         IF ($FLAG[313] OR $TIMER_FLAG[7]) AND $OUT[4039] THEN
            PREVSTEP = $APP_INT[5]
            $APP_INT[5] = 30
         ENDIF
      ;ENDFOLD
   ;ENDFOLD
   ;FOLD SCHRITT 30 -- ROB EZ1/SP1/KE1 SZ3 -- ;%{P}%MKUKATPVW,%CSTEP,%VST_NR,%P 1:SCHRITT, 2:30, 3: ROB EZ1/SP1/KE1 SZ3
      ;FOLD ;%{H}
         Case 30
      ;ENDFOLD
      ;FOLD F312 = AUS ;%{SE}%MKUKATPVW %CVW_SPS %VBOASG %P 2:F312 = AUS, 3: BOASG
         $FLAG[312] = FALSE
      ;ENDFOLD
      ;FOLD -- KF1/KW1 Ausblasen ein -- ;%{SE}%MKUKATPVW %CVW_COM %VCOMMENT %P 2:-- KF1/KW1 Ausblasen ein --, 3: VW_COMMENT
      ;ENDFOLD
      ;FOLD A835 = (F330 + !F330 & !F331 & !F332) & !F289 ;%{SE}%MKUKATPVW %CVW_SPS %VBOASG %P 2:A835 = (F330 + !F330 & !F331 & !F332) & !F289, 3: BOASG
         $OUT[835] = ($FLAG[330] OR NOT $FLAG[330] AND NOT $FLAG[331] AND NOT $FLAG[332]) AND NOT $FLAG[289]
      ;ENDFOLD
      ;FOLD A859 = (F330 + !F330 & !F331 & !F332) & F289 ;%{SE}%MKUKATPVW %CVW_SPS %VBOASG %P 2:A859 = (F330 + !F330 & !F331 & !F332) & F289, 3: BOASG
         $OUT[859] = ($FLAG[330] OR NOT $FLAG[330] AND NOT $FLAG[331] AND NOT $FLAG[332]) AND $FLAG[289]
      ;ENDFOLD
      ;FOLD A1019 = (F330 + !F330 & !F331 & !F332) & F803 ;%{SE}%MKUKATPVW %CVW_SPS %VBOASG %P 2:A1019 = (F330 + !F330 & !F331 & !F332) & F803, 3: BOASG
         $OUT[1019] = ($FLAG[330] OR NOT $FLAG[330] AND NOT $FLAG[331] AND NOT $FLAG[332]) AND $FLAG[803]
      ;ENDFOLD
      ;FOLD Schritt 31 = A4039  ;%{SE}%MKUKATPVW %CVW_SPS %VST_CON %P 2:Schritt 31 = A4039 , 3: ST_CON
         IF $OUT[4039] THEN
            PREVSTEP = $APP_INT[5]
            $APP_INT[5] = 31
         ENDIF
      ;ENDFOLD
   ;ENDFOLD
   ;FOLD SCHRITT 31 -- ROB EZ1/SP1/KE1 SZ3 -- ;%{P}%MKUKATPVW,%CSTEP,%VST_NR,%P 1:SCHRITT, 2:31, 3: ROB EZ1/SP1/KE1 SZ3
      ;FOLD ;%{H}
         Case 31
      ;ENDFOLD
      ;FOLD -- RSK Fehlerausgabe KF1/KW1 Initiator/Motor -- ;%{SE}%MKUKATPVW %CVW_COM %VCOMMENT %P 2:-- RSK Fehlerausgabe KF1/KW1 Initiator/Motor --, 3: VW_COMMENT
      ;ENDFOLD
      ;FOLD F322 = !F313 ;%{SE}%MKUKATPVW %CVW_SPS %VBOASG %P 2:F322 = !F313, 3: BOASG
         $FLAG[322] = NOT $FLAG[313]
      ;ENDFOLD
      ;FOLD T7 ( EIN ) = STOP ;%{SE}%MKUKATPVW %CVW_SPS %VTSTOP %P 2:T7 ( EIN ) = STOP, 3: TSTOP
         VW(#SET_TIME,TRUE,7,1,0)
      ;ENDFOLD
      ;FOLD A834 = !F322 & !F289 ;%{SE}%MKUKATPVW %CVW_SPS %VBOASG %P 2:A834 = !F322 & !F289, 3: BOASG
         $OUT[834] = NOT $FLAG[322] AND NOT $FLAG[289]
      ;ENDFOLD
      ;FOLD A858 = !F322 & F289 ;%{SE}%MKUKATPVW %CVW_SPS %VBOASG %P 2:A858 = !F322 & F289, 3: BOASG
         $OUT[858] = NOT $FLAG[322] AND $FLAG[289]
      ;ENDFOLD
      ;FOLD A1018 = !F322 & F803 ;%{SE}%MKUKATPVW %CVW_SPS %VBOASG %P 2:A1018 = !F322 & F803, 3: BOASG
         $OUT[1018] = NOT $FLAG[322] AND $FLAG[803]
      ;ENDFOLD
      ;FOLD Schritt 32 = !F322 & A4039  ;%{SE}%MKUKATPVW %CVW_SPS %VST_CON %P 2:Schritt 32 = !F322 & A4039 , 3: ST_CON
         IF NOT $FLAG[322] AND $OUT[4039] THEN
            PREVSTEP = $APP_INT[5]
            $APP_INT[5] = 32
         ENDIF
      ;ENDFOLD
      ;FOLD Schritt 34 = F322 & A4039  ;%{SE}%MKUKATPVW %CVW_SPS %VST_CON %P 2:Schritt 34 = F322 & A4039 , 3: ST_CON
         IF $FLAG[322] AND $OUT[4039] THEN
            PREVSTEP = $APP_INT[5]
            $APP_INT[5] = 34
         ENDIF
      ;ENDFOLD
   ;ENDFOLD
   ;FOLD SCHRITT 32 -- ROB EZ1/SP1/KE1 SZ3 -- ;%{P}%MKUKATPVW,%CSTEP,%VST_NR,%P 1:SCHRITT, 2:32, 3: ROB EZ1/SP1/KE1 SZ3
      ;FOLD ;%{H}
         Case 32
      ;ENDFOLD
      ;FOLD F312 = AUS ;%{SE}%MKUKATPVW %CVW_SPS %VBOASG %P 2:F312 = AUS, 3: BOASG
         $FLAG[312] = FALSE
      ;ENDFOLD
      ;FOLD F313 = AUS ;%{SE}%MKUKATPVW %CVW_SPS %VBOASG %P 2:F313 = AUS, 3: BOASG
         $FLAG[313] = FALSE
      ;ENDFOLD
      ;FOLD -- Umdreh. KF setzen -- ;%{SE}%MKUKATPVW %CVW_COM %VCOMMENT %P 2:-- Umdreh. KF setzen --, 3: VW_COMMENT
      ;ENDFOLD
      ;FOLD F270 = F111 & F732 ;%{SE}%MKUKATPVW %CVW_SPS %VBOASG %P 2:F270 = F111 & F732, 3: BOASG
         $FLAG[270] = $FLAG[111] AND $FLAG[732]
      ;ENDFOLD
      ;FOLD i45 ( EIN ) = i13 ;%{SE}%MKUKATPVW %CVW_SPS %VARIASG %P 2:i45 ( EIN ) = i13, 3: ARIASG
         VW(#COUNTER,TRUE,45,$COUNT_I[13])
      ;ENDFOLD
      ;FOLD i13 ( F270 ) = i43 ;%{SE}%MKUKATPVW %CVW_SPS %VARIASG %P 2:i13 ( F270 ) = i43, 3: ARIASG
         VW(#COUNTER,$FLAG[270],13,$COUNT_I[43])
      ;ENDFOLD
      ;FOLD i1 ( EIN ) = 0 ;%{SE}%MKUKATPVW %CVW_SPS %VARIASG %P 2:i1 ( EIN ) = 0, 3: ARIASG
         VW(#COUNTER,TRUE,1,0)
      ;ENDFOLD
      ;FOLD -- Ueberwachungszeit EZ1/SP1 SZ3 schliessen -- ;%{SE}%MKUKATPVW %CVW_COM %VCOMMENT %P 2:-- Ueberwachungszeit EZ1/SP1 SZ3 schliessen --, 3: VW_COMMENT
      ;ENDFOLD
      ;FOLD T9 ( EIN ) = -40[1/10Sek] ;%{SE}%MKUKATPVW %CVW_SPS %VTASG %P 2:T9 ( EIN ) = -40[1/10Sek], 3: TASG
         VW(#SET_TIME,TRUE,9,0,-40)
      ;ENDFOLD
      ;FOLD -- Ueberwachungszeit KF1/KW1 -- ;%{SE}%MKUKATPVW %CVW_COM %VCOMMENT %P 2:-- Ueberwachungszeit KF1/KW1 --, 3: VW_COMMENT
      ;ENDFOLD
      ;FOLD T7 ( EIN ) = -40[1/10Sek] ;%{SE}%MKUKATPVW %CVW_SPS %VTASG %P 2:T7 ( EIN ) = -40[1/10Sek], 3: TASG
         VW(#SET_TIME,TRUE,7,0,-40)
      ;ENDFOLD
      ;FOLD Schritt 33 = A4039  ;%{SE}%MKUKATPVW %CVW_SPS %VST_CON %P 2:Schritt 33 = A4039 , 3: ST_CON
         IF $OUT[4039] THEN
            PREVSTEP = $APP_INT[5]
            $APP_INT[5] = 33
         ENDIF
      ;ENDFOLD
   ;ENDFOLD
   ;FOLD SCHRITT 33 -- ROB EZ1/SP1/KE1 SZ3 -- ;%{P}%MKUKATPVW,%CSTEP,%VST_NR,%P 1:SCHRITT, 2:33, 3: ROB EZ1/SP1/KE1 SZ3
      ;FOLD ;%{H}
         Case 33
      ;ENDFOLD
      ;FOLD F270 = AUS ;%{SE}%MKUKATPVW %CVW_SPS %VBOASG %P 2:F270 = AUS, 3: BOASG
         $FLAG[270] = FALSE
      ;ENDFOLD
      ;FOLD -- KF1/KW1 Ausblasen -- ;%{SE}%MKUKATPVW %CVW_COM %VCOMMENT %P 2:-- KF1/KW1 Ausblasen --, 3: VW_COMMENT
      ;ENDFOLD
      ;FOLD A835 = (F330 + F331 + !F330 & !F331 & !F332) & !F289 ;%{SE}%MKUKATPVW %CVW_SPS %VBOASG %P 2:A835 = (F330 + F331 + !F330 & !F331 & !F332) & !F289, 3: BOASG
         $OUT[835] = ($FLAG[330] OR $FLAG[331] OR NOT $FLAG[330] AND NOT $FLAG[331] AND NOT $FLAG[332]) AND NOT $FLAG[289]
      ;ENDFOLD
      ;FOLD A859 = (F330 + F331 + !F330 & !F331 & !F332) & F289 ;%{SE}%MKUKATPVW %CVW_SPS %VBOASG %P 2:A859 = (F330 + F331 + !F330 & !F331 & !F332) & F289, 3: BOASG
         $OUT[859] = ($FLAG[330] OR $FLAG[331] OR NOT $FLAG[330] AND NOT $FLAG[331] AND NOT $FLAG[332]) AND $FLAG[289]
      ;ENDFOLD
      ;FOLD A1019 = (F330 + F331 + !F330 & !F331 & !F332) & F803 ;%{SE}%MKUKATPVW %CVW_SPS %VBOASG %P 2:A1019 = (F330 + F331 + !F330 & !F331 & !F332) & F803, 3: BOASG
         $OUT[1019] = ($FLAG[330] OR $FLAG[331] OR NOT $FLAG[330] AND NOT $FLAG[331] AND NOT $FLAG[332]) AND $FLAG[803]
      ;ENDFOLD
      ;FOLD -- EZ1/SP1 SZ3 schliessen -- ;%{SE}%MKUKATPVW %CVW_COM %VCOMMENT %P 2:-- EZ1/SP1 SZ3 schliessen --, 3: VW_COMMENT
      ;ENDFOLD
      ;FOLD A717 = AUS ;%{SE}%MKUKATPVW %CVW_SPS %VBOASG %P 2:A717 = AUS, 3: BOASG
         $OUT[717] = FALSE
      ;ENDFOLD
      ;FOLD A718 = EIN ;%{SE}%MKUKATPVW %CVW_SPS %VBOASG %P 2:A718 = EIN, 3: BOASG
         $OUT[718] = TRUE
      ;ENDFOLD
      ;FOLD Schritt 34 = (!E717 & E718 + T9) & A4039  ;%{SE}%MKUKATPVW %CVW_SPS %VST_CON %P 2:Schritt 34 = (!E717 & E718 + T9) & A4039 , 3: ST_CON
         IF (NOT $IN[717] AND $IN[718] OR $TIMER_FLAG[9]) AND $OUT[4039] THEN
            PREVSTEP = $APP_INT[5]
            $APP_INT[5] = 34
         ENDIF
      ;ENDFOLD
   ;ENDFOLD
   ;FOLD SCHRITT 34 -- ROB EZ1/SP1/KE1 SZ3 -- ;%{P}%MKUKATPVW,%CSTEP,%VST_NR,%P 1:SCHRITT, 2:34, 3: ROB EZ1/SP1/KE1 SZ3
      ;FOLD ;%{H}
         Case 34
      ;ENDFOLD
      ;FOLD T9 ( EIN ) = STOP ;%{SE}%MKUKATPVW %CVW_SPS %VTSTOP %P 2:T9 ( EIN ) = STOP, 3: TSTOP
         VW(#SET_TIME,TRUE,9,1,0)
      ;ENDFOLD
      ;FOLD -- RSK Fehlerausgabe Kraftaufbau -- ;%{SE}%MKUKATPVW %CVW_COM %VCOMMENT %P 2:-- RSK Fehlerausgabe Kraftaufbau --, 3: VW_COMMENT
      ;ENDFOLD
      ;FOLD F325 = T9 ;%{SE}%MKUKATPVW %CVW_SPS %VBOASG %P 2:F325 = T9, 3: BOASG
         $FLAG[325] = $TIMER_FLAG[9]
      ;ENDFOLD
      ;FOLD -- KF1/KW1 abschalten bei Fehler -- ;%{SE}%MKUKATPVW %CVW_COM %VCOMMENT %P 2:-- KF1/KW1 abschalten bei Fehler --, 3: VW_COMMENT
      ;ENDFOLD
      ;FOLD A834 = !T7 & !T9 & !F289 ;%{SE}%MKUKATPVW %CVW_SPS %VBOASG %P 2:A834 = !T7 & !T9 & !F289, 3: BOASG
         $OUT[834] = NOT $TIMER_FLAG[7] AND NOT $TIMER_FLAG[9] AND NOT $FLAG[289]
      ;ENDFOLD
      ;FOLD A858 = !T7 & !T9 & F289 ;%{SE}%MKUKATPVW %CVW_SPS %VBOASG %P 2:A858 = !T7 & !T9 & F289, 3: BOASG
         $OUT[858] = NOT $TIMER_FLAG[7] AND NOT $TIMER_FLAG[9] AND $FLAG[289]
      ;ENDFOLD
      ;FOLD A1018 = !T7 & !T9 & F803 ;%{SE}%MKUKATPVW %CVW_SPS %VBOASG %P 2:A1018 = !T7 & !T9 & F803, 3: BOASG
         $OUT[1018] = NOT $TIMER_FLAG[7] AND NOT $TIMER_FLAG[9] AND $FLAG[803]
      ;ENDFOLD
      ;FOLD -- KF1/KW1 Ausblasen -- ;%{SE}%MKUKATPVW %CVW_COM %VCOMMENT %P 2:-- KF1/KW1 Ausblasen --, 3: VW_COMMENT
      ;ENDFOLD
      ;FOLD A835 = (F330 + F331 + !F330 & !F331 & !F332) & !T9 & !F289 ;%{SE}%MKUKATPVW %CVW_SPS %VBOASG %P 2:A835 = (F330 + F331 + !F330 & !F331 & !F332) & !T9 & !F289, 3: BOASG
         $OUT[835] = ($FLAG[330] OR $FLAG[331] OR NOT $FLAG[330] AND NOT $FLAG[331] AND NOT $FLAG[332]) AND NOT $TIMER_FLAG[9] AND NOT $FLAG[289]
      ;ENDFOLD
      ;FOLD A859 = (F330 + F331 + !F330 & !F331 & !F332) & !T9 & F289 ;%{SE}%MKUKATPVW %CVW_SPS %VBOASG %P 2:A859 = (F330 + F331 + !F330 & !F331 & !F332) & !T9 & F289, 3: BOASG
         $OUT[859] = ($FLAG[330] OR $FLAG[331] OR NOT $FLAG[330] AND NOT $FLAG[331] AND NOT $FLAG[332]) AND NOT $TIMER_FLAG[9] AND $FLAG[289]
      ;ENDFOLD
      ;FOLD A1019 = (F330 + F331 + !F330 & !F331 & !F332) & !T9 & F803 ;%{SE}%MKUKATPVW %CVW_SPS %VBOASG %P 2:A1019 = (F330 + F331 + !F330 & !F331 & !F332) & !T9 & F803, 3: BOASG
         $OUT[1019] = ($FLAG[330] OR $FLAG[331] OR NOT $FLAG[330] AND NOT $FLAG[331] AND NOT $FLAG[332]) AND NOT $TIMER_FLAG[9] AND $FLAG[803]
      ;ENDFOLD
      ;FOLD -- Warte Fraesen fertig oder Timeout -- ;%{SE}%MKUKATPVW %CVW_COM %VCOMMENT %P 2:-- Warte Fraesen fertig oder Timeout --, 3: VW_COMMENT
      ;ENDFOLD
      ;FOLD Schritt 35 = (F110 & F79 + F106 & !F287 & F78 + F108 & F287 & F78 + T7 + T9) & A4039  ;%{SE}%MKUKATPVW %CVW_SPS %VST_CON %P 2:Schritt 35 = (F110 & F79 + F106 & !F287 & F78 + F108 & F287 & F78 + T7 + T9) & A4039 , 3: ST_CON
         IF ($FLAG[110] AND $FLAG[79] OR $FLAG[106] AND NOT $FLAG[287] AND $FLAG[78] OR $FLAG[108] AND $FLAG[287] AND $FLAG[78] OR $TIMER_FLAG[7] OR $TIMER_FLAG[9]) AND $OUT[4039] THEN
            PREVSTEP = $APP_INT[5]
            $APP_INT[5] = 35
         ENDIF
      ;ENDFOLD
   ;ENDFOLD
   ;FOLD SCHRITT 35 -- ROB EZ1/SP1/KE1 SZ3 -- ;%{P}%MKUKATPVW,%CSTEP,%VST_NR,%P 1:SCHRITT, 2:35, 3: ROB EZ1/SP1/KE1 SZ3
      ;FOLD ;%{H}
         Case 35
      ;ENDFOLD
      ;FOLD -- Hilfsflag SK Programmwechsel -- ;%{SE}%MKUKATPVW %CVW_COM %VCOMMENT %P 2:-- Hilfsflag SK Programmwechsel --, 3: VW_COMMENT
      ;ENDFOLD
      ;FOLD F334 = AUS ;%{SE}%MKUKATPVW %CVW_SPS %VBOASG %P 2:F334 = AUS, 3: BOASG
         $FLAG[334] = FALSE
      ;ENDFOLD
      ;FOLD t7 ( EIN ) = STOP ;%{SE}%MKUKATPVW %CVW_SPS %VTSTOP %P 2:t7 ( EIN ) = STOP, 3: TSTOP
         VW(#SET_TIME,TRUE,7,1,0)
      ;ENDFOLD
      ;FOLD -- KF1 Ausblasen -- ;%{SE}%MKUKATPVW %CVW_COM %VCOMMENT %P 2:-- KF1 Ausblasen --, 3: VW_COMMENT
      ;ENDFOLD
      ;FOLD A835 = (F330 + F331 + F332 + !F330 & !F331 & !F332) & !F289 ;%{SE}%MKUKATPVW %CVW_SPS %VBOASG %P 2:A835 = (F330 + F331 + F332 + !F330 & !F331 & !F332) & !F289, 3: BOASG
         $OUT[835] = ($FLAG[330] OR $FLAG[331] OR $FLAG[332] OR NOT $FLAG[330] AND NOT $FLAG[331] AND NOT $FLAG[332]) AND NOT $FLAG[289]
      ;ENDFOLD
      ;FOLD A859 = (F330 + F331 + F332 + !F330 & !F331 & !F332) & F289 ;%{SE}%MKUKATPVW %CVW_SPS %VBOASG %P 2:A859 = (F330 + F331 + F332 + !F330 & !F331 & !F332) & F289, 3: BOASG
         $OUT[859] = ($FLAG[330] OR $FLAG[331] OR $FLAG[332] OR NOT $FLAG[330] AND NOT $FLAG[331] AND NOT $FLAG[332]) AND $FLAG[289]
      ;ENDFOLD
      ;FOLD A1019 = (F330 + F331 + F332 + !F330 & !F331 & !F332) & F803 ;%{SE}%MKUKATPVW %CVW_SPS %VBOASG %P 2:A1019 = (F330 + F331 + F332 + !F330 & !F331 & !F332) & F803, 3: BOASG
         $OUT[1019] = ($FLAG[330] OR $FLAG[331] OR $FLAG[332] OR NOT $FLAG[330] AND NOT $FLAG[331] AND NOT $FLAG[332]) AND $FLAG[803]
      ;ENDFOLD
      ;FOLD -- KF Ausblasen Ausschaltverzoegerung starten -- ;%{SE}%MKUKATPVW %CVW_COM %VCOMMENT %P 2:-- KF Ausblasen Ausschaltverzoegerung starten --, 3: VW_COMMENT
      ;ENDFOLD
      ;FOLD F736 = EIN ;%{SE}%MKUKATPVW %CVW_SPS %VBOASG %P 2:F736 = EIN, 3: BOASG
         $FLAG[736] = TRUE
      ;ENDFOLD
      ;FOLD -- EZ1/SP1 SZ3 oeffnen -- ;%{SE}%MKUKATPVW %CVW_COM %VCOMMENT %P 2:-- EZ1/SP1 SZ3 oeffnen --, 3: VW_COMMENT
      ;ENDFOLD
      ;FOLD A719 = AUS ;%{SE}%MKUKATPVW %CVW_SPS %VBOASG %P 2:A719 = AUS, 3: BOASG
         $OUT[719] = FALSE
      ;ENDFOLD
      ;FOLD A718 = AUS ;%{SE}%MKUKATPVW %CVW_SPS %VBOASG %P 2:A718 = AUS, 3: BOASG
         $OUT[718] = FALSE
      ;ENDFOLD
      ;FOLD A717 = EIN ;%{SE}%MKUKATPVW %CVW_SPS %VBOASG %P 2:A717 = EIN, 3: BOASG
         $OUT[717] = TRUE
      ;ENDFOLD
      ;FOLD -- RSK Sammelstoerung -- ;%{SE}%MKUKATPVW %CVW_COM %VCOMMENT %P 2:-- RSK Sammelstoerung --, 3: VW_COMMENT
      ;ENDFOLD
      ;FOLD F329 = T7 + T9 ;%{SE}%MKUKATPVW %CVW_SPS %VBOASG %P 2:F329 = T7 + T9, 3: BOASG
         $FLAG[329] = $TIMER_FLAG[7] OR $TIMER_FLAG[9]
      ;ENDFOLD
      ;FOLD -- Hilfsflag Startfraesen -- ;%{SE}%MKUKATPVW %CVW_COM %VCOMMENT %P 2:-- Hilfsflag Startfraesen --, 3: VW_COMMENT
      ;ENDFOLD
      ;FOLD F108 = (F108 & F78 + F110 & F79) & F287 ;%{SE}%MKUKATPVW %CVW_SPS %VBOASG %P 2:F108 = (F108 & F78 + F110 & F79) & F287, 3: BOASG
         $FLAG[108] = ($FLAG[108] AND $FLAG[78] OR $FLAG[110] AND $FLAG[79]) AND $FLAG[287]
      ;ENDFOLD
      ;FOLD F110 = !F130 & F110 + F130 & F287 & F110 ;%{SE}%MKUKATPVW %CVW_SPS %VBOASG %P 2:F110 = !F130 & F110 + F130 & F287 & F110, 3: BOASG
         $FLAG[110] = NOT $FLAG[130] AND $FLAG[110] OR $FLAG[130] AND $FLAG[287] AND $FLAG[110]
      ;ENDFOLD
      ;FOLD F287 = F78 + F79 & F130 ;%{SE}%MKUKATPVW %CVW_SPS %VBOASG %P 2:F287 = F78 + F79 & F130, 3: BOASG
         $FLAG[287] = $FLAG[78] OR $FLAG[79] AND $FLAG[130]
      ;ENDFOLD
      ;FOLD -- Neues Fraesprogramm und Zaehler ruecksetzen -- ;%{SE}%MKUKATPVW %CVW_COM %VCOMMENT %P 2:-- Neues Fraesprogramm und Zaehler ruecksetzen --, 3: VW_COMMENT
      ;ENDFOLD
      ;FOLD F270 = F108 & F732 ;%{SE}%MKUKATPVW %CVW_SPS %VBOASG %P 2:F270 = F108 & F732, 3: BOASG
         $FLAG[270] = $FLAG[108] AND $FLAG[732]
      ;ENDFOLD
      ;FOLD bin3 ( F732 ) = 38 ;%{SE}%MKUKATPVW %CVW_SPS %VARIASG %P 2:bin3 ( F732 ) = 38, 3: ARIASG
         VW(#BINOUT,$FLAG[732],3,38)
      ;ENDFOLD
      ;FOLD i13 ( F270 ) = i45 ;%{SE}%MKUKATPVW %CVW_SPS %VARIASG %P 2:i13 ( F270 ) = i45, 3: ARIASG
         VW(#COUNTER,$FLAG[270],13,$COUNT_I[45])
      ;ENDFOLD
      ;FOLD -- Wiederholung beim Startfraesen -- ;%{SE}%MKUKATPVW %CVW_COM %VCOMMENT %P 2:-- Wiederholung beim Startfraesen --, 3: VW_COMMENT
      ;ENDFOLD
      ;FOLD Schritt 32 = E717 & !E718 & (F78 & !F108 + F79 & F130 & !F108) & !F329 & A4039  ;%{SE}%MKUKATPVW %CVW_SPS %VST_CON %P 2:Schritt 32 = E717 & !E718 & (F78 & !F108 + F79 & F130 & !F108) & !F329 & A4039 , 3: ST_CON
         IF $IN[717] AND NOT $IN[718] AND ($FLAG[78] AND NOT $FLAG[108] OR $FLAG[79] AND $FLAG[130] AND NOT $FLAG[108]) AND NOT $FLAG[329] AND $OUT[4039] THEN
            PREVSTEP = $APP_INT[5]
            $APP_INT[5] = 32
         ENDIF
      ;ENDFOLD
      ;FOLD -- Weiter wenn Fraesen fertig -- ;%{SE}%MKUKATPVW %CVW_COM %VCOMMENT %P 2:-- Weiter wenn Fraesen fertig --, 3: VW_COMMENT
      ;ENDFOLD
      ;FOLD Schritt 36 = E717 & !E718 & (F79 & F110 & (!F130 + F108) + F78 & F108 + F329) & A4039  ;%{SE}%MKUKATPVW %CVW_SPS %VST_CON %P 2:Schritt 36 = E717 & !E718 & (F79 & F110 & (!F130 + F108) + F78 & F108 + F329) & A4039 , 3: ST_CON
         IF $IN[717] AND NOT $IN[718] AND ($FLAG[79] AND $FLAG[110] AND (NOT $FLAG[130] OR $FLAG[108]) OR $FLAG[78] AND $FLAG[108] OR $FLAG[329]) AND $OUT[4039] THEN
            PREVSTEP = $APP_INT[5]
            $APP_INT[5] = 36
         ENDIF
      ;ENDFOLD
      ;FOLD -- Weiter bei Fehler -- ;%{SE}%MKUKATPVW %CVW_COM %VCOMMENT %P 2:-- Weiter bei Fehler --, 3: VW_COMMENT
      ;ENDFOLD
      ;FOLD Schritt 38 = F325 & (E26 + E27) & A4039  ;%{SE}%MKUKATPVW %CVW_SPS %VST_CON %P 2:Schritt 38 = F325 & (E26 + E27) & A4039 , 3: ST_CON
         IF $FLAG[325] AND ($IN[26] OR $IN[27]) AND $OUT[4039] THEN
            PREVSTEP = $APP_INT[5]
            $APP_INT[5] = 38
         ENDIF
      ;ENDFOLD
   ;ENDFOLD
   ;FOLD SCHRITT 36 -- ROB EZ1/SP1/KE1 SZ3 -- ;%{P}%MKUKATPVW,%CSTEP,%VST_NR,%P 1:SCHRITT, 2:36, 3: ROB EZ1/SP1/KE1 SZ3
      ;FOLD ;%{H}
         Case 36
      ;ENDFOLD
      ;FOLD F270 = AUS ;%{SE}%MKUKATPVW %CVW_SPS %VBOASG %P 2:F270 = AUS, 3: BOASG
         $FLAG[270] = FALSE
      ;ENDFOLD
      ;FOLD A717 = AUS ;%{SE}%MKUKATPVW %CVW_SPS %VBOASG %P 2:A717 = AUS, 3: BOASG
         $OUT[717] = FALSE
      ;ENDFOLD
      ;FOLD -- KF1/KW1 abschalten -- ;%{SE}%MKUKATPVW %CVW_COM %VCOMMENT %P 2:-- KF1/KW1 abschalten --, 3: VW_COMMENT
      ;ENDFOLD
      ;FOLD A834 = AUS ;%{SE}%MKUKATPVW %CVW_SPS %VBOASG %P 2:A834 = AUS, 3: BOASG
         $OUT[834] = FALSE
      ;ENDFOLD
      ;FOLD A858 = AUS ;%{SE}%MKUKATPVW %CVW_SPS %VBOASG %P 2:A858 = AUS, 3: BOASG
         $OUT[858] = FALSE
      ;ENDFOLD
      ;FOLD A1018 = AUS ;%{SE}%MKUKATPVW %CVW_SPS %VBOASG %P 2:A1018 = AUS, 3: BOASG
         $OUT[1018] = FALSE
      ;ENDFOLD
      ;FOLD bin3 ( !F329 ) = 3 ;%{SE}%MKUKATPVW %CVW_SPS %VARIASG %P 2:bin3 ( !F329 ) = 3, 3: ARIASG
         VW(#BINOUT,NOT $FLAG[329],3,3)
      ;ENDFOLD
      ;FOLD -- Wartezeit Programmwechsel SK -- ;%{SE}%MKUKATPVW %CVW_COM %VCOMMENT %P 2:-- Wartezeit Programmwechsel SK --, 3: VW_COMMENT
      ;ENDFOLD
      ;FOLD T8 ( !F334 ) = -2[1/10Sek] ;%{SE}%MKUKATPVW %CVW_SPS %VTASG %P 2:T8 ( !F334 ) = -2[1/10Sek], 3: TASG
         VW(#SET_TIME,NOT $FLAG[334],8,0,-2)
      ;ENDFOLD
      ;FOLD -- Hilfsflag SK Programmwechsel -- ;%{SE}%MKUKATPVW %CVW_COM %VCOMMENT %P 2:-- Hilfsflag SK Programmwechsel --, 3: VW_COMMENT
      ;ENDFOLD
      ;FOLD F334 = EIN ;%{SE}%MKUKATPVW %CVW_SPS %VBOASG %P 2:F334 = EIN, 3: BOASG
         $FLAG[334] = TRUE
      ;ENDFOLD
      ;FOLD Schritt 37 = T8 & A4039  ;%{SE}%MKUKATPVW %CVW_SPS %VST_CON %P 2:Schritt 37 = T8 & A4039 , 3: ST_CON
         IF $TIMER_FLAG[8] AND $OUT[4039] THEN
            PREVSTEP = $APP_INT[5]
            $APP_INT[5] = 37
         ENDIF
      ;ENDFOLD
   ;ENDFOLD
   ;FOLD SCHRITT 37 -- ROB EZ1/SP1/KE1 SZ3 -- ;%{P}%MKUKATPVW,%CSTEP,%VST_NR,%P 1:SCHRITT, 2:37, 3: ROB EZ1/SP1/KE1 SZ3
      ;FOLD ;%{H}
         Case 37
      ;ENDFOLD
      ;FOLD -- Hilfsflag SK Programmwechsel -- ;%{SE}%MKUKATPVW %CVW_COM %VCOMMENT %P 2:-- Hilfsflag SK Programmwechsel --, 3: VW_COMMENT
      ;ENDFOLD
      ;FOLD F334 = AUS ;%{SE}%MKUKATPVW %CVW_SPS %VBOASG %P 2:F334 = AUS, 3: BOASG
         $FLAG[334] = FALSE
      ;ENDFOLD
      ;FOLD -- Quitt. Fraesen SK1 -- ;%{SE}%MKUKATPVW %CVW_COM %VCOMMENT %P 2:-- Quitt. Fraesen SK1 --, 3: VW_COMMENT
      ;ENDFOLD
      ;FOLD A786 = (!F329 & !F322 & !F830) + (F830 & A786) ;%{SE}%MKUKATPVW %CVW_SPS %VBOASG %P 2:A786 = (!F329 & !F322 & !F830) + (F830 & A786), 3: BOASG
         $OUT[786] = (NOT $FLAG[329] AND NOT $FLAG[322] AND NOT $FLAG[830]) OR ($FLAG[830] AND $OUT[786])
      ;ENDFOLD
      ;FOLD A722 = (!F329 & !F322 & F830) + (!F830 & A722) ;%{SE}%MKUKATPVW %CVW_SPS %VBOASG %P 2:A722 = (!F329 & !F322 & F830) + (!F830 & A722), 3: BOASG
         $OUT[722] = (NOT $FLAG[329] AND NOT $FLAG[322] AND $FLAG[830]) OR (NOT $FLAG[830] AND $OUT[722])
      ;ENDFOLD
      ;FOLD Schritt 38 = (!F830 & !E786 & E787 & !E788 + F830 & !E722 & E724 & !E723 + F329) & A4039  ;%{SE}%MKUKATPVW %CVW_SPS %VST_CON %P 2:Schritt 38 = (!F830 & !E786 & E787 & !E788 + F830 & !E722 & E724 & !E723 + F329) & A4039 , 3: ST_CON
         IF (NOT $FLAG[830] AND NOT $IN[786] AND $IN[787] AND NOT $IN[788] OR $FLAG[830] AND NOT $IN[722] AND $IN[724] AND NOT $IN[723] OR $FLAG[329]) AND $OUT[4039] THEN
            PREVSTEP = $APP_INT[5]
            $APP_INT[5] = 38
         ENDIF
      ;ENDFOLD
   ;ENDFOLD
   ;FOLD SCHRITT 38 -- ROB EZ1/SP1/KE1 SZ3 # Ende -- ;%{P}%MKUKATPVW,%CSTEP,%VST_NR,%P 1:SCHRITT, 2:38, 3: ROB EZ1/SP1/KE1 SZ3 # Ende
      ;FOLD ;%{H}
         Case 38
      ;ENDFOLD
      ;FOLD F270 = AUS ;%{SE}%MKUKATPVW %CVW_SPS %VBOASG %P 2:F270 = AUS, 3: BOASG
         $FLAG[270] = FALSE
      ;ENDFOLD
      ;FOLD -- KF1/KW1 Ausblasen -- ;%{SE}%MKUKATPVW %CVW_COM %VCOMMENT %P 2:-- KF1/KW1 Ausblasen --, 3: VW_COMMENT
      ;ENDFOLD
      ;FOLD A835 = (F330 + F331 + F332) & F736 ;%{SE}%MKUKATPVW %CVW_SPS %VBOASG %P 2:A835 = (F330 + F331 + F332) & F736, 3: BOASG
         $OUT[835] = ($FLAG[330] OR $FLAG[331] OR $FLAG[332]) AND $FLAG[736]
      ;ENDFOLD
      ;FOLD A859 = (F330 + F331 + F332) & F736 & F289 ;%{SE}%MKUKATPVW %CVW_SPS %VBOASG %P 2:A859 = (F330 + F331 + F332) & F736 & F289, 3: BOASG
         $OUT[859] = ($FLAG[330] OR $FLAG[331] OR $FLAG[332]) AND $FLAG[736] AND $FLAG[289]
      ;ENDFOLD
      ;FOLD A1019 = (F330 + F331 + F332) & F736 & F803 ;%{SE}%MKUKATPVW %CVW_SPS %VBOASG %P 2:A1019 = (F330 + F331 + F332) & F736 & F803, 3: BOASG
         $OUT[1019] = ($FLAG[330] OR $FLAG[331] OR $FLAG[332]) AND $FLAG[736] AND $FLAG[803]
      ;ENDFOLD
      ;FOLD F91 = (!E786 & E787 & !E788 & !F830 + !E722 & E724 & !E723 & F830) & !F322 & !F325 & !F329 ;%{SE}%MKUKATPVW %CVW_SPS %VBOASG %P 2:F91 = (!E786 & E787 & !E788 & !F830 + !E722 & E724 & !E723 & F830) & !F322 & !F325 & !F329, 3: BOASG
         $FLAG[91] = (NOT $IN[786] AND $IN[787] AND NOT $IN[788] AND NOT $FLAG[830] OR NOT $IN[722] AND $IN[724] AND NOT $IN[723] AND $FLAG[830]) AND NOT $FLAG[322] AND NOT $FLAG[325] AND NOT $FLAG[329]
      ;ENDFOLD
      ;FOLD Schritt 27 = (F322 + F325 + F329) & (E26 + E27) & A4039  ;%{SE}%MKUKATPVW %CVW_SPS %VST_CON %P 2:Schritt 27 = (F322 + F325 + F329) & (E26 + E27) & A4039 , 3: ST_CON
         IF ($FLAG[322] OR $FLAG[325] OR $FLAG[329]) AND ($IN[26] OR $IN[27]) AND $OUT[4039] THEN
            PREVSTEP = $APP_INT[5]
            $APP_INT[5] = 27
         ENDIF
      ;ENDFOLD
      ;FOLD Schritt 1 = F91 & !F322 & !F325 & !F329 & A4039  ;%{SE}%MKUKATPVW %CVW_SPS %VST_CON %P 2:Schritt 1 = F91 & !F322 & !F325 & !F329 & A4039 , 3: ST_CON
         IF $FLAG[91] AND NOT $FLAG[322] AND NOT $FLAG[325] AND NOT $FLAG[329] AND $OUT[4039] THEN
            PREVSTEP = $APP_INT[5]
            $APP_INT[5] = 1
         ENDIF
      ;ENDFOLD
   ;ENDFOLD
   ;FOLD SCHRITT 39 -- ROB EZ1/SP1/KE1 SZ4 # Start -- ;%{P}%MKUKATPVW,%CSTEP,%VST_NR,%P 1:SCHRITT, 2:39, 3: ROB EZ1/SP1/KE1 SZ4 # Start
      ;FOLD ;%{H}
         Case 39
      ;ENDFOLD
      ;FOLD -- RSK gestartet -- ;%{SE}%MKUKATPVW %CVW_COM %VCOMMENT %P 2:-- RSK gestartet --, 3: VW_COMMENT
      ;ENDFOLD
      ;FOLD F321 = AUS ;%{SE}%MKUKATPVW %CVW_SPS %VBOASG %P 2:F321 = AUS, 3: BOASG
         $FLAG[321] = FALSE
      ;ENDFOLD
      ;FOLD F322 = AUS ;%{SE}%MKUKATPVW %CVW_SPS %VBOASG %P 2:F322 = AUS, 3: BOASG
         $FLAG[322] = FALSE
      ;ENDFOLD
      ;FOLD F323 = AUS ;%{SE}%MKUKATPVW %CVW_SPS %VBOASG %P 2:F323 = AUS, 3: BOASG
         $FLAG[323] = FALSE
      ;ENDFOLD
      ;FOLD F324 = AUS ;%{SE}%MKUKATPVW %CVW_SPS %VBOASG %P 2:F324 = AUS, 3: BOASG
         $FLAG[324] = FALSE
      ;ENDFOLD
      ;FOLD F325 = AUS ;%{SE}%MKUKATPVW %CVW_SPS %VBOASG %P 2:F325 = AUS, 3: BOASG
         $FLAG[325] = FALSE
      ;ENDFOLD
      ;FOLD F327 = AUS ;%{SE}%MKUKATPVW %CVW_SPS %VBOASG %P 2:F327 = AUS, 3: BOASG
         $FLAG[327] = FALSE
      ;ENDFOLD
      ;FOLD F329 = AUS ;%{SE}%MKUKATPVW %CVW_SPS %VBOASG %P 2:F329 = AUS, 3: BOASG
         $FLAG[329] = FALSE
      ;ENDFOLD
      ;FOLD -- EZ1/SP1 SZ4 Zaehler -- ;%{SE}%MKUKATPVW %CVW_COM %VCOMMENT %P 2:-- EZ1/SP1 SZ4 Zaehler --, 3: VW_COMMENT
      ;ENDFOLD
      ;FOLD F112 = AUS ;%{SE}%MKUKATPVW %CVW_SPS %VBOASG %P 2:F112 = AUS, 3: BOASG
         $FLAG[112] = FALSE
      ;ENDFOLD
      ;FOLD F113 = AUS ;%{SE}%MKUKATPVW %CVW_SPS %VBOASG %P 2:F113 = AUS, 3: BOASG
         $FLAG[113] = FALSE
      ;ENDFOLD
      ;FOLD F114 = AUS ;%{SE}%MKUKATPVW %CVW_SPS %VBOASG %P 2:F114 = AUS, 3: BOASG
         $FLAG[114] = FALSE
      ;ENDFOLD
      ;FOLD F115 = AUS ;%{SE}%MKUKATPVW %CVW_SPS %VBOASG %P 2:F115 = AUS, 3: BOASG
         $FLAG[115] = FALSE
      ;ENDFOLD
      ;FOLD F116 = AUS ;%{SE}%MKUKATPVW %CVW_SPS %VBOASG %P 2:F116 = AUS, 3: BOASG
         $FLAG[116] = FALSE
      ;ENDFOLD
      ;FOLD F117 = AUS ;%{SE}%MKUKATPVW %CVW_SPS %VBOASG %P 2:F117 = AUS, 3: BOASG
         $FLAG[117] = FALSE
      ;ENDFOLD
      ;FOLD -- Hilfsflags Funktionstest KF Motor -- ;%{SE}%MKUKATPVW %CVW_COM %VCOMMENT %P 2:-- Hilfsflags Funktionstest KF Motor --, 3: VW_COMMENT
      ;ENDFOLD
      ;FOLD F312 = AUS ;%{SE}%MKUKATPVW %CVW_SPS %VBOASG %P 2:F312 = AUS, 3: BOASG
         $FLAG[312] = FALSE
      ;ENDFOLD
      ;FOLD F313 = AUS ;%{SE}%MKUKATPVW %CVW_SPS %VBOASG %P 2:F313 = AUS, 3: BOASG
         $FLAG[313] = FALSE
      ;ENDFOLD
      ;FOLD -- Rob. EZ1/SP1 SZ4 beim Fraesen -- ;%{SE}%MKUKATPVW %CVW_COM %VCOMMENT %P 2:-- Rob. EZ1/SP1 SZ4 beim Fraesen --, 3: VW_COMMENT
      ;ENDFOLD
      ;FOLD A116 = EIN ;%{SE}%MKUKATPVW %CVW_SPS %VBOASG %P 2:A116 = EIN, 3: BOASG
         $OUT[116] = TRUE
      ;ENDFOLD
      ;FOLD A130 = EIN ;%{SE}%MKUKATPVW %CVW_SPS %VBOASG %P 2:A130 = EIN, 3: BOASG
         $OUT[130] = TRUE
      ;ENDFOLD
      ;FOLD -- Quitt. Fraesen SK1 AUS -- ;%{SE}%MKUKATPVW %CVW_COM %VCOMMENT %P 2:-- Quitt. Fraesen SK1 AUS --, 3: VW_COMMENT
      ;ENDFOLD
      ;FOLD A786 = F830 & A786 ;%{SE}%MKUKATPVW %CVW_SPS %VBOASG %P 2:A786 = F830 & A786, 3: BOASG
         $OUT[786] = $FLAG[830] AND $OUT[786]
      ;ENDFOLD
      ;FOLD A722 = !F830 & A722 ;%{SE}%MKUKATPVW %CVW_SPS %VBOASG %P 2:A722 = !F830 & A722, 3: BOASG
         $OUT[722] = NOT $FLAG[830] AND $OUT[722]
      ;ENDFOLD
      ;FOLD -- Ueberwachungszeit KF1/KW1 -- ;%{SE}%MKUKATPVW %CVW_COM %VCOMMENT %P 2:-- Ueberwachungszeit KF1/KW1 --, 3: VW_COMMENT
      ;ENDFOLD
      ;FOLD t7 ( EIN ) = -30[1/10Sek] ;%{SE}%MKUKATPVW %CVW_SPS %VTASG %P 2:t7 ( EIN ) = -30[1/10Sek], 3: TASG
         VW(#SET_TIME,TRUE,7,0,-30)
      ;ENDFOLD
      ;FOLD Schritt 40 = A4039  ;%{SE}%MKUKATPVW %CVW_SPS %VST_CON %P 2:Schritt 40 = A4039 , 3: ST_CON
         IF $OUT[4039] THEN
            PREVSTEP = $APP_INT[5]
            $APP_INT[5] = 40
         ENDIF
      ;ENDFOLD
   ;ENDFOLD
   ;FOLD SCHRITT 40 -- ROB EZ1/SP1/KE1 SZ4 -- ;%{P}%MKUKATPVW,%CSTEP,%VST_NR,%P 1:SCHRITT, 2:40, 3: ROB EZ1/SP1/KE1 SZ4
      ;FOLD ;%{H}
         Case 40
      ;ENDFOLD
      ;FOLD -- KF1/KW1 einschalten -- ;%{SE}%MKUKATPVW %CVW_COM %VCOMMENT %P 2:-- KF1/KW1 einschalten --, 3: VW_COMMENT
      ;ENDFOLD
      ;FOLD i1 (EIN) = 0 ;%{SE}%MKUKATPVW %CVW_SPS %VARIASG %P 2:i1 (EIN) = 0, 3: ARIASG
         VW(#COUNTER,TRUE,1,0)
      ;ENDFOLD
      ;FOLD A834 = !F289 ;%{SE}%MKUKATPVW %CVW_SPS %VBOASG %P 2:A834 = !F289, 3: BOASG
         $OUT[834] = NOT $FLAG[289]
      ;ENDFOLD
      ;FOLD A858 = F289 ;%{SE}%MKUKATPVW %CVW_SPS %VBOASG %P 2:A858 = F289, 3: BOASG
         $OUT[858] = $FLAG[289]
      ;ENDFOLD
      ;FOLD A1018 = F803 ;%{SE}%MKUKATPVW %CVW_SPS %VBOASG %P 2:A1018 = F803, 3: BOASG
         $OUT[1018] = $FLAG[803]
      ;ENDFOLD
      ;FOLD Schritt 41 = A4039  ;%{SE}%MKUKATPVW %CVW_SPS %VST_CON %P 2:Schritt 41 = A4039 , 3: ST_CON
         IF $OUT[4039] THEN
            PREVSTEP = $APP_INT[5]
            $APP_INT[5] = 41
         ENDIF
      ;ENDFOLD
   ;ENDFOLD
   ;FOLD SCHRITT 41 -- ROB EZ1/SP1/KE1 SZ4 -- ;%{P}%MKUKATPVW,%CSTEP,%VST_NR,%P 1:SCHRITT, 2:41, 3: ROB EZ1/SP1/KE1 SZ4
      ;FOLD ;%{H}
         Case 41
      ;ENDFOLD
      ;FOLD -- Funktionstest KF Motor -- ;%{SE}%MKUKATPVW %CVW_COM %VCOMMENT %P 2:-- Funktionstest KF Motor --, 3: VW_COMMENT
      ;ENDFOLD
      ;FOLD F312 = EIN ;%{SE}%MKUKATPVW %CVW_SPS %VBOASG %P 2:F312 = EIN, 3: BOASG
         $FLAG[312] = TRUE
      ;ENDFOLD
      ;FOLD F313 = i1 > 2 ;%{SE}%MKUKATPVW %CVW_SPS %VBOCMP %P 2:F313 = i1 > 2, 3: BOCMP
         $FLAG[313] = $COUNT_I[1] > 2
      ;ENDFOLD
      ;FOLD Schritt 42 = (F313 + T7) & A4039  ;%{SE}%MKUKATPVW %CVW_SPS %VST_CON %P 2:Schritt 42 = (F313 + T7) & A4039 , 3: ST_CON
         IF ($FLAG[313] OR $TIMER_FLAG[7]) AND $OUT[4039] THEN
            PREVSTEP = $APP_INT[5]
            $APP_INT[5] = 42
         ENDIF
      ;ENDFOLD
   ;ENDFOLD
   ;FOLD SCHRITT 42 -- ROB EZ1/SP1/KE1 SZ4 -- ;%{P}%MKUKATPVW,%CSTEP,%VST_NR,%P 1:SCHRITT, 2:42, 3: ROB EZ1/SP1/KE1 SZ4
      ;FOLD ;%{H}
         Case 42
      ;ENDFOLD
      ;FOLD F312 = AUS ;%{SE}%MKUKATPVW %CVW_SPS %VBOASG %P 2:F312 = AUS, 3: BOASG
         $FLAG[312] = FALSE
      ;ENDFOLD
      ;FOLD -- KF1/KW1 Ausblasen ein -- ;%{SE}%MKUKATPVW %CVW_COM %VCOMMENT %P 2:-- KF1/KW1 Ausblasen ein --, 3: VW_COMMENT
      ;ENDFOLD
      ;FOLD A835 = (F330 + !F330 & !F331 & !F332) & !F289 ;%{SE}%MKUKATPVW %CVW_SPS %VBOASG %P 2:A835 = (F330 + !F330 & !F331 & !F332) & !F289, 3: BOASG
         $OUT[835] = ($FLAG[330] OR NOT $FLAG[330] AND NOT $FLAG[331] AND NOT $FLAG[332]) AND NOT $FLAG[289]
      ;ENDFOLD
      ;FOLD A859 = (F330 + !F330 & !F331 & !F332) & F289 ;%{SE}%MKUKATPVW %CVW_SPS %VBOASG %P 2:A859 = (F330 + !F330 & !F331 & !F332) & F289, 3: BOASG
         $OUT[859] = ($FLAG[330] OR NOT $FLAG[330] AND NOT $FLAG[331] AND NOT $FLAG[332]) AND $FLAG[289]
      ;ENDFOLD
      ;FOLD A1019 = (F330 + !F330 & !F331 & !F332) & F803 ;%{SE}%MKUKATPVW %CVW_SPS %VBOASG %P 2:A1019 = (F330 + !F330 & !F331 & !F332) & F803, 3: BOASG
         $OUT[1019] = ($FLAG[330] OR NOT $FLAG[330] AND NOT $FLAG[331] AND NOT $FLAG[332]) AND $FLAG[803]
      ;ENDFOLD
      ;FOLD Schritt 43 = A4039  ;%{SE}%MKUKATPVW %CVW_SPS %VST_CON %P 2:Schritt 43 = A4039 , 3: ST_CON
         IF $OUT[4039] THEN
            PREVSTEP = $APP_INT[5]
            $APP_INT[5] = 43
         ENDIF
      ;ENDFOLD
   ;ENDFOLD
   ;FOLD SCHRITT 43 -- ROB EZ1/SP1/KE1 SZ4 -- ;%{P}%MKUKATPVW,%CSTEP,%VST_NR,%P 1:SCHRITT, 2:43, 3: ROB EZ1/SP1/KE1 SZ4
      ;FOLD ;%{H}
         Case 43
      ;ENDFOLD
      ;FOLD -- RSK Fehlerausgabe KF1/KW1 Initiator/Motor -- ;%{SE}%MKUKATPVW %CVW_COM %VCOMMENT %P 2:-- RSK Fehlerausgabe KF1/KW1 Initiator/Motor --, 3: VW_COMMENT
      ;ENDFOLD
      ;FOLD F322 = !F313 ;%{SE}%MKUKATPVW %CVW_SPS %VBOASG %P 2:F322 = !F313, 3: BOASG
         $FLAG[322] = NOT $FLAG[313]
      ;ENDFOLD
      ;FOLD T7 ( EIN ) = STOP ;%{SE}%MKUKATPVW %CVW_SPS %VTSTOP %P 2:T7 ( EIN ) = STOP, 3: TSTOP
         VW(#SET_TIME,TRUE,7,1,0)
      ;ENDFOLD
      ;FOLD A834 = !F322 & !F289 ;%{SE}%MKUKATPVW %CVW_SPS %VBOASG %P 2:A834 = !F322 & !F289, 3: BOASG
         $OUT[834] = NOT $FLAG[322] AND NOT $FLAG[289]
      ;ENDFOLD
      ;FOLD A858 = !F322 & F289 ;%{SE}%MKUKATPVW %CVW_SPS %VBOASG %P 2:A858 = !F322 & F289, 3: BOASG
         $OUT[858] = NOT $FLAG[322] AND $FLAG[289]
      ;ENDFOLD
      ;FOLD A1018 = !F322 & F803 ;%{SE}%MKUKATPVW %CVW_SPS %VBOASG %P 2:A1018 = !F322 & F803, 3: BOASG
         $OUT[1018] = NOT $FLAG[322] AND $FLAG[803]
      ;ENDFOLD
      ;FOLD Schritt 44 = !F322 & A4039  ;%{SE}%MKUKATPVW %CVW_SPS %VST_CON %P 2:Schritt 44 = !F322 & A4039 , 3: ST_CON
         IF NOT $FLAG[322] AND $OUT[4039] THEN
            PREVSTEP = $APP_INT[5]
            $APP_INT[5] = 44
         ENDIF
      ;ENDFOLD
      ;FOLD Schritt 46 = F322 & A4039  ;%{SE}%MKUKATPVW %CVW_SPS %VST_CON %P 2:Schritt 46 = F322 & A4039 , 3: ST_CON
         IF $FLAG[322] AND $OUT[4039] THEN
            PREVSTEP = $APP_INT[5]
            $APP_INT[5] = 46
         ENDIF
      ;ENDFOLD
   ;ENDFOLD
   ;FOLD SCHRITT 44 -- ROB EZ1/SP1/KE1 SZ4 -- ;%{P}%MKUKATPVW,%CSTEP,%VST_NR,%P 1:SCHRITT, 2:44, 3: ROB EZ1/SP1/KE1 SZ4
      ;FOLD ;%{H}
         Case 44
      ;ENDFOLD
      ;FOLD F312 = AUS ;%{SE}%MKUKATPVW %CVW_SPS %VBOASG %P 2:F312 = AUS, 3: BOASG
         $FLAG[312] = FALSE
      ;ENDFOLD
      ;FOLD F313 = AUS ;%{SE}%MKUKATPVW %CVW_SPS %VBOASG %P 2:F313 = AUS, 3: BOASG
         $FLAG[313] = FALSE
      ;ENDFOLD
      ;FOLD -- Umdreh. KF setzen -- ;%{SE}%MKUKATPVW %CVW_COM %VCOMMENT %P 2:-- Umdreh. KF setzen --, 3: VW_COMMENT
      ;ENDFOLD
      ;FOLD F270 = F117 & F732 ;%{SE}%MKUKATPVW %CVW_SPS %VBOASG %P 2:F270 = F117 & F732, 3: BOASG
         $FLAG[270] = $FLAG[117] AND $FLAG[732]
      ;ENDFOLD
      ;FOLD i45 ( EIN ) = i16 ;%{SE}%MKUKATPVW %CVW_SPS %VARIASG %P 2:i45 ( EIN ) = i16, 3: ARIASG
         VW(#COUNTER,TRUE,45,$COUNT_I[16])
      ;ENDFOLD
      ;FOLD i16 ( F270 ) = i43 ;%{SE}%MKUKATPVW %CVW_SPS %VARIASG %P 2:i16 ( F270 ) = i43, 3: ARIASG
         VW(#COUNTER,$FLAG[270],16,$COUNT_I[43])
      ;ENDFOLD
      ;FOLD i1 ( EIN ) = 0 ;%{SE}%MKUKATPVW %CVW_SPS %VARIASG %P 2:i1 ( EIN ) = 0, 3: ARIASG
         VW(#COUNTER,TRUE,1,0)
      ;ENDFOLD
      ;FOLD -- Ueberwachungszeit EZ1/SP1/KE1 SZ4 schliessen -- ;%{SE}%MKUKATPVW %CVW_COM %VCOMMENT %P 2:-- Ueberwachungszeit EZ1/SP1/KE1 SZ4 schliessen --, 3: VW_COMMENT
      ;ENDFOLD
      ;FOLD T9 ( EIN ) = -40[1/10Sek] ;%{SE}%MKUKATPVW %CVW_SPS %VTASG %P 2:T9 ( EIN ) = -40[1/10Sek], 3: TASG
         VW(#SET_TIME,TRUE,9,0,-40)
      ;ENDFOLD
      ;FOLD -- Ueberwachungszeit KF1 -- ;%{SE}%MKUKATPVW %CVW_COM %VCOMMENT %P 2:-- Ueberwachungszeit KF1 --, 3: VW_COMMENT
      ;ENDFOLD
      ;FOLD T7 ( EIN ) = -40[1/10Sek] ;%{SE}%MKUKATPVW %CVW_SPS %VTASG %P 2:T7 ( EIN ) = -40[1/10Sek], 3: TASG
         VW(#SET_TIME,TRUE,7,0,-40)
      ;ENDFOLD
      ;FOLD Schritt 45 = A4039  ;%{SE}%MKUKATPVW %CVW_SPS %VST_CON %P 2:Schritt 45 = A4039 , 3: ST_CON
         IF $OUT[4039] THEN
            PREVSTEP = $APP_INT[5]
            $APP_INT[5] = 45
         ENDIF
      ;ENDFOLD
   ;ENDFOLD
   ;FOLD SCHRITT 45 -- ROB EZ1/SP1/KE1 SZ4 -- ;%{P}%MKUKATPVW,%CSTEP,%VST_NR,%P 1:SCHRITT, 2:45, 3: ROB EZ1/SP1/KE1 SZ4
      ;FOLD ;%{H}
         Case 45
      ;ENDFOLD
      ;FOLD F270 = AUS ;%{SE}%MKUKATPVW %CVW_SPS %VBOASG %P 2:F270 = AUS, 3: BOASG
         $FLAG[270] = FALSE
      ;ENDFOLD
      ;FOLD -- KF1/KW1 Ausblasen -- ;%{SE}%MKUKATPVW %CVW_COM %VCOMMENT %P 2:-- KF1/KW1 Ausblasen --, 3: VW_COMMENT
      ;ENDFOLD
      ;FOLD A835 = (F330 + F331 + !F330 & !F331 & !F332) & !F289 ;%{SE}%MKUKATPVW %CVW_SPS %VBOASG %P 2:A835 = (F330 + F331 + !F330 & !F331 & !F332) & !F289, 3: BOASG
         $OUT[835] = ($FLAG[330] OR $FLAG[331] OR NOT $FLAG[330] AND NOT $FLAG[331] AND NOT $FLAG[332]) AND NOT $FLAG[289]
      ;ENDFOLD
      ;FOLD A859 = (F330 + F331 + !F330 & !F331 & !F332) & F289 ;%{SE}%MKUKATPVW %CVW_SPS %VBOASG %P 2:A859 = (F330 + F331 + !F330 & !F331 & !F332) & F289, 3: BOASG
         $OUT[859] = ($FLAG[330] OR $FLAG[331] OR NOT $FLAG[330] AND NOT $FLAG[331] AND NOT $FLAG[332]) AND $FLAG[289]
      ;ENDFOLD
      ;FOLD A1019 = (F330 + F331 + !F330 & !F331 & !F332) & F803 ;%{SE}%MKUKATPVW %CVW_SPS %VBOASG %P 2:A1019 = (F330 + F331 + !F330 & !F331 & !F332) & F803, 3: BOASG
         $OUT[1019] = ($FLAG[330] OR $FLAG[331] OR NOT $FLAG[330] AND NOT $FLAG[331] AND NOT $FLAG[332]) AND $FLAG[803]
      ;ENDFOLD
      ;FOLD -- EZ1/SP1 SZ4 schliessen -- ;%{SE}%MKUKATPVW %CVW_COM %VCOMMENT %P 2:-- EZ1/SP1 SZ4 schliessen --, 3: VW_COMMENT
      ;ENDFOLD
      ;FOLD A717 = AUS ;%{SE}%MKUKATPVW %CVW_SPS %VBOASG %P 2:A717 = AUS, 3: BOASG
         $OUT[717] = FALSE
      ;ENDFOLD
      ;FOLD A718 = EIN ;%{SE}%MKUKATPVW %CVW_SPS %VBOASG %P 2:A718 = EIN, 3: BOASG
         $OUT[718] = TRUE
      ;ENDFOLD
      ;FOLD Schritt 46 = (!E717 & E718 + T9) & A4039  ;%{SE}%MKUKATPVW %CVW_SPS %VST_CON %P 2:Schritt 46 = (!E717 & E718 + T9) & A4039 , 3: ST_CON
         IF (NOT $IN[717] AND $IN[718] OR $TIMER_FLAG[9]) AND $OUT[4039] THEN
            PREVSTEP = $APP_INT[5]
            $APP_INT[5] = 46
         ENDIF
      ;ENDFOLD
   ;ENDFOLD
   ;FOLD SCHRITT 46 -- ROB EZ1/SP1/KE1 SZ4 -- ;%{P}%MKUKATPVW,%CSTEP,%VST_NR,%P 1:SCHRITT, 2:46, 3: ROB EZ1/SP1/KE1 SZ4
      ;FOLD ;%{H}
         Case 46
      ;ENDFOLD
      ;FOLD T9 ( EIN ) = STOP ;%{SE}%MKUKATPVW %CVW_SPS %VTSTOP %P 2:T9 ( EIN ) = STOP, 3: TSTOP
         VW(#SET_TIME,TRUE,9,1,0)
      ;ENDFOLD
      ;FOLD -- RSK Fehlerausgabe Kraftaufbau -- ;%{SE}%MKUKATPVW %CVW_COM %VCOMMENT %P 2:-- RSK Fehlerausgabe Kraftaufbau --, 3: VW_COMMENT
      ;ENDFOLD
      ;FOLD F325 = T9 ;%{SE}%MKUKATPVW %CVW_SPS %VBOASG %P 2:F325 = T9, 3: BOASG
         $FLAG[325] = $TIMER_FLAG[9]
      ;ENDFOLD
      ;FOLD -- KF1/KW1 abschalten bei Fehler -- ;%{SE}%MKUKATPVW %CVW_COM %VCOMMENT %P 2:-- KF1/KW1 abschalten bei Fehler --, 3: VW_COMMENT
      ;ENDFOLD
      ;FOLD A834 = !T7 & !T9 & !F289 ;%{SE}%MKUKATPVW %CVW_SPS %VBOASG %P 2:A834 = !T7 & !T9 & !F289, 3: BOASG
         $OUT[834] = NOT $TIMER_FLAG[7] AND NOT $TIMER_FLAG[9] AND NOT $FLAG[289]
      ;ENDFOLD
      ;FOLD A858 = !T7 & !T9 & F289 ;%{SE}%MKUKATPVW %CVW_SPS %VBOASG %P 2:A858 = !T7 & !T9 & F289, 3: BOASG
         $OUT[858] = NOT $TIMER_FLAG[7] AND NOT $TIMER_FLAG[9] AND $FLAG[289]
      ;ENDFOLD
      ;FOLD A1018 = !T7 & !T9 & F803 ;%{SE}%MKUKATPVW %CVW_SPS %VBOASG %P 2:A1018 = !T7 & !T9 & F803, 3: BOASG
         $OUT[1018] = NOT $TIMER_FLAG[7] AND NOT $TIMER_FLAG[9] AND $FLAG[803]
      ;ENDFOLD
      ;FOLD -- KF1/KW1 Ausblasen -- ;%{SE}%MKUKATPVW %CVW_COM %VCOMMENT %P 2:-- KF1/KW1 Ausblasen --, 3: VW_COMMENT
      ;ENDFOLD
      ;FOLD A835 = (F330 + F331 + !F330 & !F331 & !F332) & !T9 & !F289 ;%{SE}%MKUKATPVW %CVW_SPS %VBOASG %P 2:A835 = (F330 + F331 + !F330 & !F331 & !F332) & !T9 & !F289, 3: BOASG
         $OUT[835] = ($FLAG[330] OR $FLAG[331] OR NOT $FLAG[330] AND NOT $FLAG[331] AND NOT $FLAG[332]) AND NOT $TIMER_FLAG[9] AND NOT $FLAG[289]
      ;ENDFOLD
      ;FOLD A859 = (F330 + F331 + !F330 & !F331 & !F332) & !T9 & F289 ;%{SE}%MKUKATPVW %CVW_SPS %VBOASG %P 2:A859 = (F330 + F331 + !F330 & !F331 & !F332) & !T9 & F289, 3: BOASG
         $OUT[859] = ($FLAG[330] OR $FLAG[331] OR NOT $FLAG[330] AND NOT $FLAG[331] AND NOT $FLAG[332]) AND NOT $TIMER_FLAG[9] AND $FLAG[289]
      ;ENDFOLD
      ;FOLD A1019 = (F330 + F331 + !F330 & !F331 & !F332) & !T9 & F803 ;%{SE}%MKUKATPVW %CVW_SPS %VBOASG %P 2:A1019 = (F330 + F331 + !F330 & !F331 & !F332) & !T9 & F803, 3: BOASG
         $OUT[1019] = ($FLAG[330] OR $FLAG[331] OR NOT $FLAG[330] AND NOT $FLAG[331] AND NOT $FLAG[332]) AND NOT $TIMER_FLAG[9] AND $FLAG[803]
      ;ENDFOLD
      ;FOLD -- Warte Fraesen fertig oder Timeout -- ;%{SE}%MKUKATPVW %CVW_COM %VCOMMENT %P 2:-- Warte Fraesen fertig oder Timeout --, 3: VW_COMMENT
      ;ENDFOLD
      ;FOLD Schritt 47 = (F116 & F79 + F112 & !F287 & F78 + F114 & F287 & F78 + T7 + T9) & A4039  ;%{SE}%MKUKATPVW %CVW_SPS %VST_CON %P 2:Schritt 47 = (F116 & F79 + F112 & !F287 & F78 + F114 & F287 & F78 + T7 + T9) & A4039 , 3: ST_CON
         IF ($FLAG[116] AND $FLAG[79] OR $FLAG[112] AND NOT $FLAG[287] AND $FLAG[78] OR $FLAG[114] AND $FLAG[287] AND $FLAG[78] OR $TIMER_FLAG[7] OR $TIMER_FLAG[9]) AND $OUT[4039] THEN
            PREVSTEP = $APP_INT[5]
            $APP_INT[5] = 47
         ENDIF
      ;ENDFOLD
   ;ENDFOLD
   ;FOLD SCHRITT 47 -- ROB EZ1/SP1/KE1 SZ4 -- ;%{P}%MKUKATPVW,%CSTEP,%VST_NR,%P 1:SCHRITT, 2:47, 3: ROB EZ1/SP1/KE1 SZ4
      ;FOLD ;%{H}
         Case 47
      ;ENDFOLD
      ;FOLD -- Hilfsflag SK Programmwechsel -- ;%{SE}%MKUKATPVW %CVW_COM %VCOMMENT %P 2:-- Hilfsflag SK Programmwechsel --, 3: VW_COMMENT
      ;ENDFOLD
      ;FOLD F334 = AUS ;%{SE}%MKUKATPVW %CVW_SPS %VBOASG %P 2:F334 = AUS, 3: BOASG
         $FLAG[334] = FALSE
      ;ENDFOLD
      ;FOLD t7 ( EIN ) = STOP ;%{SE}%MKUKATPVW %CVW_SPS %VTSTOP %P 2:t7 ( EIN ) = STOP, 3: TSTOP
         VW(#SET_TIME,TRUE,7,1,0)
      ;ENDFOLD
      ;FOLD -- KF1/KW1 Ausblasen -- ;%{SE}%MKUKATPVW %CVW_COM %VCOMMENT %P 2:-- KF1/KW1 Ausblasen --, 3: VW_COMMENT
      ;ENDFOLD
      ;FOLD A835 = (F330 + F331 + F332 + !F330 & !F331 & !F332) & !F289 ;%{SE}%MKUKATPVW %CVW_SPS %VBOASG %P 2:A835 = (F330 + F331 + F332 + !F330 & !F331 & !F332) & !F289, 3: BOASG
         $OUT[835] = ($FLAG[330] OR $FLAG[331] OR $FLAG[332] OR NOT $FLAG[330] AND NOT $FLAG[331] AND NOT $FLAG[332]) AND NOT $FLAG[289]
      ;ENDFOLD
      ;FOLD A859 = (F330 + F331 + F332 + !F330 & !F331 & !F332) & F289 ;%{SE}%MKUKATPVW %CVW_SPS %VBOASG %P 2:A859 = (F330 + F331 + F332 + !F330 & !F331 & !F332) & F289, 3: BOASG
         $OUT[859] = ($FLAG[330] OR $FLAG[331] OR $FLAG[332] OR NOT $FLAG[330] AND NOT $FLAG[331] AND NOT $FLAG[332]) AND $FLAG[289]
      ;ENDFOLD
      ;FOLD A1019 = (F330 + F331 + F332 + !F330 & !F331 & !F332) & F803 ;%{SE}%MKUKATPVW %CVW_SPS %VBOASG %P 2:A1019 = (F330 + F331 + F332 + !F330 & !F331 & !F332) & F803, 3: BOASG
         $OUT[1019] = ($FLAG[330] OR $FLAG[331] OR $FLAG[332] OR NOT $FLAG[330] AND NOT $FLAG[331] AND NOT $FLAG[332]) AND $FLAG[803]
      ;ENDFOLD
      ;FOLD -- KF Ausblasen Ausschaltverzoegerung starten -- ;%{SE}%MKUKATPVW %CVW_COM %VCOMMENT %P 2:-- KF Ausblasen Ausschaltverzoegerung starten --, 3: VW_COMMENT
      ;ENDFOLD
      ;FOLD F736 = EIN ;%{SE}%MKUKATPVW %CVW_SPS %VBOASG %P 2:F736 = EIN, 3: BOASG
         $FLAG[736] = TRUE
      ;ENDFOLD
      ;FOLD -- EZ1/SP1 SZ4 oeffnen -- ;%{SE}%MKUKATPVW %CVW_COM %VCOMMENT %P 2:-- EZ1/SP1 SZ4 oeffnen --, 3: VW_COMMENT
      ;ENDFOLD
      ;FOLD A719 = AUS ;%{SE}%MKUKATPVW %CVW_SPS %VBOASG %P 2:A719 = AUS, 3: BOASG
         $OUT[719] = FALSE
      ;ENDFOLD
      ;FOLD A718 = AUS ;%{SE}%MKUKATPVW %CVW_SPS %VBOASG %P 2:A718 = AUS, 3: BOASG
         $OUT[718] = FALSE
      ;ENDFOLD
      ;FOLD A717 = EIN ;%{SE}%MKUKATPVW %CVW_SPS %VBOASG %P 2:A717 = EIN, 3: BOASG
         $OUT[717] = TRUE
      ;ENDFOLD
      ;FOLD -- RSK Sammelstoerung -- ;%{SE}%MKUKATPVW %CVW_COM %VCOMMENT %P 2:-- RSK Sammelstoerung --, 3: VW_COMMENT
      ;ENDFOLD
      ;FOLD F329 = T7 + T9 ;%{SE}%MKUKATPVW %CVW_SPS %VBOASG %P 2:F329 = T7 + T9, 3: BOASG
         $FLAG[329] = $TIMER_FLAG[7] OR $TIMER_FLAG[9]
      ;ENDFOLD
      ;FOLD -- Hilfsflag Startfraesen -- ;%{SE}%MKUKATPVW %CVW_COM %VCOMMENT %P 2:-- Hilfsflag Startfraesen --, 3: VW_COMMENT
      ;ENDFOLD
      ;FOLD F114 = (F114 & F78 + F116 & F79) & F287 ;%{SE}%MKUKATPVW %CVW_SPS %VBOASG %P 2:F114 = (F114 & F78 + F116 & F79) & F287, 3: BOASG
         $FLAG[114] = ($FLAG[114] AND $FLAG[78] OR $FLAG[116] AND $FLAG[79]) AND $FLAG[287]
      ;ENDFOLD
      ;FOLD F116 = !F130 & F116 + F130 & F287 & F116 ;%{SE}%MKUKATPVW %CVW_SPS %VBOASG %P 2:F116 = !F130 & F116 + F130 & F287 & F116, 3: BOASG
         $FLAG[116] = NOT $FLAG[130] AND $FLAG[116] OR $FLAG[130] AND $FLAG[287] AND $FLAG[116]
      ;ENDFOLD
      ;FOLD F287 = F78 + F79 & F130 ;%{SE}%MKUKATPVW %CVW_SPS %VBOASG %P 2:F287 = F78 + F79 & F130, 3: BOASG
         $FLAG[287] = $FLAG[78] OR $FLAG[79] AND $FLAG[130]
      ;ENDFOLD
      ;FOLD -- Neues Fraesprogramm und Zaehler ruecksetzen -- ;%{SE}%MKUKATPVW %CVW_COM %VCOMMENT %P 2:-- Neues Fraesprogramm und Zaehler ruecksetzen --, 3: VW_COMMENT
      ;ENDFOLD
      ;FOLD F270 = F114 & F732 ;%{SE}%MKUKATPVW %CVW_SPS %VBOASG %P 2:F270 = F114 & F732, 3: BOASG
         $FLAG[270] = $FLAG[114] AND $FLAG[732]
      ;ENDFOLD
      ;FOLD bin3 ( F732 ) = 39 ;%{SE}%MKUKATPVW %CVW_SPS %VARIASG %P 2:bin3 ( F732 ) = 39, 3: ARIASG
         VW(#BINOUT,$FLAG[732],3,39)
      ;ENDFOLD
      ;FOLD i16 ( F270 ) = i45 ;%{SE}%MKUKATPVW %CVW_SPS %VARIASG %P 2:i16 ( F270 ) = i45, 3: ARIASG
         VW(#COUNTER,$FLAG[270],16,$COUNT_I[45])
      ;ENDFOLD
      ;FOLD -- Wiederholung beim Startfraesen -- ;%{SE}%MKUKATPVW %CVW_COM %VCOMMENT %P 2:-- Wiederholung beim Startfraesen --, 3: VW_COMMENT
      ;ENDFOLD
      ;FOLD Schritt 44 = E717 & !E718 & (F78 & !F114 + F79 & F130 & !F114) & !F329 & A4039  ;%{SE}%MKUKATPVW %CVW_SPS %VST_CON %P 2:Schritt 44 = E717 & !E718 & (F78 & !F114 + F79 & F130 & !F114) & !F329 & A4039 , 3: ST_CON
         IF $IN[717] AND NOT $IN[718] AND ($FLAG[78] AND NOT $FLAG[114] OR $FLAG[79] AND $FLAG[130] AND NOT $FLAG[114]) AND NOT $FLAG[329] AND $OUT[4039] THEN
            PREVSTEP = $APP_INT[5]
            $APP_INT[5] = 44
         ENDIF
      ;ENDFOLD
      ;FOLD -- Weiter wenn Fraesen fertig -- ;%{SE}%MKUKATPVW %CVW_COM %VCOMMENT %P 2:-- Weiter wenn Fraesen fertig --, 3: VW_COMMENT
      ;ENDFOLD
      ;FOLD Schritt 48 = E717 & !E718 & (F79 & F116 & (!F130 + F114) + F78 & F114 + F329) & A4039  ;%{SE}%MKUKATPVW %CVW_SPS %VST_CON %P 2:Schritt 48 = E717 & !E718 & (F79 & F116 & (!F130 + F114) + F78 & F114 + F329) & A4039 , 3: ST_CON
         IF $IN[717] AND NOT $IN[718] AND ($FLAG[79] AND $FLAG[116] AND (NOT $FLAG[130] OR $FLAG[114]) OR $FLAG[78] AND $FLAG[114] OR $FLAG[329]) AND $OUT[4039] THEN
            PREVSTEP = $APP_INT[5]
            $APP_INT[5] = 48
         ENDIF
      ;ENDFOLD
      ;FOLD -- Weiter bei Fehler -- ;%{SE}%MKUKATPVW %CVW_COM %VCOMMENT %P 2:-- Weiter bei Fehler --, 3: VW_COMMENT
      ;ENDFOLD
      ;FOLD Schritt 50 = F325 & (E26 + E27) & A4039  ;%{SE}%MKUKATPVW %CVW_SPS %VST_CON %P 2:Schritt 50 = F325 & (E26 + E27) & A4039 , 3: ST_CON
         IF $FLAG[325] AND ($IN[26] OR $IN[27]) AND $OUT[4039] THEN
            PREVSTEP = $APP_INT[5]
            $APP_INT[5] = 50
         ENDIF
      ;ENDFOLD
   ;ENDFOLD
   ;FOLD SCHRITT 48 -- ROB EZ1/SP1/KE1 SZ4 -- ;%{P}%MKUKATPVW,%CSTEP,%VST_NR,%P 1:SCHRITT, 2:48, 3: ROB EZ1/SP1/KE1 SZ4
      ;FOLD ;%{H}
         Case 48
      ;ENDFOLD
      ;FOLD F270 = AUS ;%{SE}%MKUKATPVW %CVW_SPS %VBOASG %P 2:F270 = AUS, 3: BOASG
         $FLAG[270] = FALSE
      ;ENDFOLD
      ;FOLD A717 = AUS ;%{SE}%MKUKATPVW %CVW_SPS %VBOASG %P 2:A717 = AUS, 3: BOASG
         $OUT[717] = FALSE
      ;ENDFOLD
      ;FOLD -- KF1/KW1 abschalten -- ;%{SE}%MKUKATPVW %CVW_COM %VCOMMENT %P 2:-- KF1/KW1 abschalten --, 3: VW_COMMENT
      ;ENDFOLD
      ;FOLD A834 = AUS ;%{SE}%MKUKATPVW %CVW_SPS %VBOASG %P 2:A834 = AUS, 3: BOASG
         $OUT[834] = FALSE
      ;ENDFOLD
      ;FOLD A858 = AUS ;%{SE}%MKUKATPVW %CVW_SPS %VBOASG %P 2:A858 = AUS, 3: BOASG
         $OUT[858] = FALSE
      ;ENDFOLD
      ;FOLD A1018 = AUS ;%{SE}%MKUKATPVW %CVW_SPS %VBOASG %P 2:A1018 = AUS, 3: BOASG
         $OUT[1018] = FALSE
      ;ENDFOLD
      ;FOLD bin3 ( !F329 ) = 4 ;%{SE}%MKUKATPVW %CVW_SPS %VARIASG %P 2:bin3 ( !F329 ) = 4, 3: ARIASG
         VW(#BINOUT,NOT $FLAG[329],3,4)
      ;ENDFOLD
      ;FOLD -- Wartezeit Programmwechsel SK -- ;%{SE}%MKUKATPVW %CVW_COM %VCOMMENT %P 2:-- Wartezeit Programmwechsel SK --, 3: VW_COMMENT
      ;ENDFOLD
      ;FOLD T8 ( !F334 ) = -2[1/10Sek] ;%{SE}%MKUKATPVW %CVW_SPS %VTASG %P 2:T8 ( !F334 ) = -2[1/10Sek], 3: TASG
         VW(#SET_TIME,NOT $FLAG[334],8,0,-2)
      ;ENDFOLD
      ;FOLD -- Hilfsflag SK Programmwechsel -- ;%{SE}%MKUKATPVW %CVW_COM %VCOMMENT %P 2:-- Hilfsflag SK Programmwechsel --, 3: VW_COMMENT
      ;ENDFOLD
      ;FOLD F334 = EIN ;%{SE}%MKUKATPVW %CVW_SPS %VBOASG %P 2:F334 = EIN, 3: BOASG
         $FLAG[334] = TRUE
      ;ENDFOLD
      ;FOLD Schritt 49 = T8 & A4039  ;%{SE}%MKUKATPVW %CVW_SPS %VST_CON %P 2:Schritt 49 = T8 & A4039 , 3: ST_CON
         IF $TIMER_FLAG[8] AND $OUT[4039] THEN
            PREVSTEP = $APP_INT[5]
            $APP_INT[5] = 49
         ENDIF
      ;ENDFOLD
   ;ENDFOLD
   ;FOLD SCHRITT 49 -- ROB EZ1/SP1/KE1 SZ4 -- ;%{P}%MKUKATPVW,%CSTEP,%VST_NR,%P 1:SCHRITT, 2:49, 3: ROB EZ1/SP1/KE1 SZ4
      ;FOLD ;%{H}
         Case 49
      ;ENDFOLD
      ;FOLD -- Hilfsflag SK Programmwechsel -- ;%{SE}%MKUKATPVW %CVW_COM %VCOMMENT %P 2:-- Hilfsflag SK Programmwechsel --, 3: VW_COMMENT
      ;ENDFOLD
      ;FOLD F334 = AUS ;%{SE}%MKUKATPVW %CVW_SPS %VBOASG %P 2:F334 = AUS, 3: BOASG
         $FLAG[334] = FALSE
      ;ENDFOLD
      ;FOLD -- Quitt. Fraesen SK1 -- ;%{SE}%MKUKATPVW %CVW_COM %VCOMMENT %P 2:-- Quitt. Fraesen SK1 --, 3: VW_COMMENT
      ;ENDFOLD
      ;FOLD A786 = (!F329 & !F322 & !F830) + (F830 & A786) ;%{SE}%MKUKATPVW %CVW_SPS %VBOASG %P 2:A786 = (!F329 & !F322 & !F830) + (F830 & A786), 3: BOASG
         $OUT[786] = (NOT $FLAG[329] AND NOT $FLAG[322] AND NOT $FLAG[830]) OR ($FLAG[830] AND $OUT[786])
      ;ENDFOLD
      ;FOLD A722 = (!F329 & !F322 & F830) + (!F830 & A722) ;%{SE}%MKUKATPVW %CVW_SPS %VBOASG %P 2:A722 = (!F329 & !F322 & F830) + (!F830 & A722), 3: BOASG
         $OUT[722] = (NOT $FLAG[329] AND NOT $FLAG[322] AND $FLAG[830]) OR (NOT $FLAG[830] AND $OUT[722])
      ;ENDFOLD
      ;FOLD Schritt 50 = (!F830 & !E786 & E787 & !E788 + F830 & !E722 & E724 & !E723 + F329) & A4039  ;%{SE}%MKUKATPVW %CVW_SPS %VST_CON %P 2:Schritt 50 = (!F830 & !E786 & E787 & !E788 + F830 & !E722 & E724 & !E723 + F329) & A4039 , 3: ST_CON
         IF (NOT $FLAG[830] AND NOT $IN[786] AND $IN[787] AND NOT $IN[788] OR $FLAG[830] AND NOT $IN[722] AND $IN[724] AND NOT $IN[723] OR $FLAG[329]) AND $OUT[4039] THEN
            PREVSTEP = $APP_INT[5]
            $APP_INT[5] = 50
         ENDIF
      ;ENDFOLD
   ;ENDFOLD
   ;FOLD SCHRITT 50 -- ROB EZ1/SP1/KE1 SZ4 # Ende -- ;%{P}%MKUKATPVW,%CSTEP,%VST_NR,%P 1:SCHRITT, 2:50, 3: ROB EZ1/SP1/KE1 SZ4 # Ende
      ;FOLD ;%{H}
         Case 50
      ;ENDFOLD
      ;FOLD F270 = AUS ;%{SE}%MKUKATPVW %CVW_SPS %VBOASG %P 2:F270 = AUS, 3: BOASG
         $FLAG[270] = FALSE
      ;ENDFOLD
      ;FOLD -- KF1/KW1 Ausblasen -- ;%{SE}%MKUKATPVW %CVW_COM %VCOMMENT %P 2:-- KF1/KW1 Ausblasen --, 3: VW_COMMENT
      ;ENDFOLD
      ;FOLD A835 = (F330 + F331 + F332) & F736 ;%{SE}%MKUKATPVW %CVW_SPS %VBOASG %P 2:A835 = (F330 + F331 + F332) & F736, 3: BOASG
         $OUT[835] = ($FLAG[330] OR $FLAG[331] OR $FLAG[332]) AND $FLAG[736]
      ;ENDFOLD
      ;FOLD A859 = (F330 + F331 + F332) & F736 & F289 ;%{SE}%MKUKATPVW %CVW_SPS %VBOASG %P 2:A859 = (F330 + F331 + F332) & F736 & F289, 3: BOASG
         $OUT[859] = ($FLAG[330] OR $FLAG[331] OR $FLAG[332]) AND $FLAG[736] AND $FLAG[289]
      ;ENDFOLD
      ;FOLD A1019 = (F330 + F331 + F332) & F736 & F803 ;%{SE}%MKUKATPVW %CVW_SPS %VBOASG %P 2:A1019 = (F330 + F331 + F332) & F736 & F803, 3: BOASG
         $OUT[1019] = ($FLAG[330] OR $FLAG[331] OR $FLAG[332]) AND $FLAG[736] AND $FLAG[803]
      ;ENDFOLD
      ;FOLD F91 = (!E786 & E787 & !E788 & !F830 + !E722 & E724 & !E723 & F830) & !F322 & !F325 & !F329 ;%{SE}%MKUKATPVW %CVW_SPS %VBOASG %P 2:F91 = (!E786 & E787 & !E788 & !F830 + !E722 & E724 & !E723 & F830) & !F322 & !F325 & !F329, 3: BOASG
         $FLAG[91] = (NOT $IN[786] AND $IN[787] AND NOT $IN[788] AND NOT $FLAG[830] OR NOT $IN[722] AND $IN[724] AND NOT $IN[723] AND $FLAG[830]) AND NOT $FLAG[322] AND NOT $FLAG[325] AND NOT $FLAG[329]
      ;ENDFOLD
      ;FOLD Schritt 39 = (F322 + F325 + F329) & (E26 + E27) & A4039  ;%{SE}%MKUKATPVW %CVW_SPS %VST_CON %P 2:Schritt 39 = (F322 + F325 + F329) & (E26 + E27) & A4039 , 3: ST_CON
         IF ($FLAG[322] OR $FLAG[325] OR $FLAG[329]) AND ($IN[26] OR $IN[27]) AND $OUT[4039] THEN
            PREVSTEP = $APP_INT[5]
            $APP_INT[5] = 39
         ENDIF
      ;ENDFOLD
      ;FOLD Schritt 1 = F91 & !F322 & !F325 & !F329 & A4039  ;%{SE}%MKUKATPVW %CVW_SPS %VST_CON %P 2:Schritt 1 = F91 & !F322 & !F325 & !F329 & A4039 , 3: ST_CON
         IF $FLAG[91] AND NOT $FLAG[322] AND NOT $FLAG[325] AND NOT $FLAG[329] AND $OUT[4039] THEN
            PREVSTEP = $APP_INT[5]
            $APP_INT[5] = 1
         ENDIF
      ;ENDFOLD
   ;ENDFOLD
   ;FOLD SCHRITT 51 -- STAT EZ1/SP1/KE1 # Start-- ;%{P}%MKUKATPVW,%CSTEP,%VST_NR,%P 1:SCHRITT, 2:51, 3: STAT EZ1/SP1/KE1 # Start
      ;FOLD ;%{H}
         Case 51
      ;ENDFOLD
      ;FOLD -- RSK gestartet -- ;%{SE}%MKUKATPVW %CVW_COM %VCOMMENT %P 2:-- RSK gestartet --, 3: VW_COMMENT
      ;ENDFOLD
      ;FOLD F122 = AUS ;%{SE}%MKUKATPVW %CVW_SPS %VBOASG %P 2:F122 = AUS, 3: BOASG
         $FLAG[122] = FALSE
      ;ENDFOLD
      ;FOLD F321 = AUS ;%{SE}%MKUKATPVW %CVW_SPS %VBOASG %P 2:F321 = AUS, 3: BOASG
         $FLAG[321] = FALSE
      ;ENDFOLD
      ;FOLD F322 = AUS ;%{SE}%MKUKATPVW %CVW_SPS %VBOASG %P 2:F322 = AUS, 3: BOASG
         $FLAG[322] = FALSE
      ;ENDFOLD
      ;FOLD F323 = AUS ;%{SE}%MKUKATPVW %CVW_SPS %VBOASG %P 2:F323 = AUS, 3: BOASG
         $FLAG[323] = FALSE
      ;ENDFOLD
      ;FOLD F324 = AUS ;%{SE}%MKUKATPVW %CVW_SPS %VBOASG %P 2:F324 = AUS, 3: BOASG
         $FLAG[324] = FALSE
      ;ENDFOLD
      ;FOLD F325 = AUS ;%{SE}%MKUKATPVW %CVW_SPS %VBOASG %P 2:F325 = AUS, 3: BOASG
         $FLAG[325] = FALSE
      ;ENDFOLD
      ;FOLD F326 = AUS ;%{SE}%MKUKATPVW %CVW_SPS %VBOASG %P 2:F326 = AUS, 3: BOASG
         $FLAG[326] = FALSE
      ;ENDFOLD
      ;FOLD F327 = AUS ;%{SE}%MKUKATPVW %CVW_SPS %VBOASG %P 2:F327 = AUS, 3: BOASG
         $FLAG[327] = FALSE
      ;ENDFOLD
      ;FOLD F329 = AUS ;%{SE}%MKUKATPVW %CVW_SPS %VBOASG %P 2:F329 = AUS, 3: BOASG
         $FLAG[329] = FALSE
      ;ENDFOLD
      ;FOLD -- EZ1/SP1/KE1 SZ1 Zaehler -- ;%{SE}%MKUKATPVW %CVW_COM %VCOMMENT %P 2:-- EZ1/SP1/KE1 SZ1 Zaehler --, 3: VW_COMMENT
      ;ENDFOLD
      ;FOLD F94 = AUS ;%{SE}%MKUKATPVW %CVW_SPS %VBOASG %P 2:F94 = AUS, 3: BOASG
         $FLAG[94] = FALSE
      ;ENDFOLD
      ;FOLD F95 = AUS ;%{SE}%MKUKATPVW %CVW_SPS %VBOASG %P 2:F95 = AUS, 3: BOASG
         $FLAG[95] = FALSE
      ;ENDFOLD
      ;FOLD F96 = AUS ;%{SE}%MKUKATPVW %CVW_SPS %VBOASG %P 2:F96 = AUS, 3: BOASG
         $FLAG[96] = FALSE
      ;ENDFOLD
      ;FOLD F97 = AUS ;%{SE}%MKUKATPVW %CVW_SPS %VBOASG %P 2:F97 = AUS, 3: BOASG
         $FLAG[97] = FALSE
      ;ENDFOLD
      ;FOLD F98 = AUS ;%{SE}%MKUKATPVW %CVW_SPS %VBOASG %P 2:F98 = AUS, 3: BOASG
         $FLAG[98] = FALSE
      ;ENDFOLD
      ;FOLD F99 = AUS ;%{SE}%MKUKATPVW %CVW_SPS %VBOASG %P 2:F99 = AUS, 3: BOASG
         $FLAG[99] = FALSE
      ;ENDFOLD
      ;FOLD -- Hilfsflags Funktionstest KF Motor -- ;%{SE}%MKUKATPVW %CVW_COM %VCOMMENT %P 2:-- Hilfsflags Funktionstest KF Motor --, 3: VW_COMMENT
      ;ENDFOLD
      ;FOLD F312 = AUS ;%{SE}%MKUKATPVW %CVW_SPS %VBOASG %P 2:F312 = AUS, 3: BOASG
         $FLAG[312] = FALSE
      ;ENDFOLD
      ;FOLD F313 = AUS ;%{SE}%MKUKATPVW %CVW_SPS %VBOASG %P 2:F313 = AUS, 3: BOASG
         $FLAG[313] = FALSE
      ;ENDFOLD
      ;FOLD bin1 ( EIN ) = 31 ;%{SE}%MKUKATPVW %CVW_SPS %VARIASG %P 2:bin1 ( EIN ) = 31, 3: ARIASG
         VW(#BINOUT,TRUE,1,31)
      ;ENDFOLD
      ;FOLD bin3 ( EIN ) = 31 ;%{SE}%MKUKATPVW %CVW_SPS %VARIASG %P 2:bin3 ( EIN ) = 31, 3: ARIASG
         VW(#BINOUT,TRUE,3,31)
      ;ENDFOLD
      ;FOLD -- Wartezeit Programmwechsel SK -- ;%{SE}%MKUKATPVW %CVW_COM %VCOMMENT %P 2:-- Wartezeit Programmwechsel SK --, 3: VW_COMMENT
      ;ENDFOLD
      ;FOLD T8 ( !F334 ) = -2[1/10Sek] ;%{SE}%MKUKATPVW %CVW_SPS %VTASG %P 2:T8 ( !F334 ) = -2[1/10Sek], 3: TASG
         VW(#SET_TIME,NOT $FLAG[334],8,0,-2)
      ;ENDFOLD
      ;FOLD -- Hilfsflag SK Programmwechsel -- ;%{SE}%MKUKATPVW %CVW_COM %VCOMMENT %P 2:-- Hilfsflag SK Programmwechsel --, 3: VW_COMMENT
      ;ENDFOLD
      ;FOLD F334 = EIN ;%{SE}%MKUKATPVW %CVW_SPS %VBOASG %P 2:F334 = EIN, 3: BOASG
         $FLAG[334] = TRUE
      ;ENDFOLD
      ;FOLD -- Stat. EZ1/SP1/KE1 SZ1 beim Fraesen -- ;%{SE}%MKUKATPVW %CVW_COM %VCOMMENT %P 2:-- Stat. EZ1/SP1/KE1 SZ1 beim Fraesen --, 3: VW_COMMENT
      ;ENDFOLD
      ;FOLD A116 = EIN ;%{SE}%MKUKATPVW %CVW_SPS %VBOASG %P 2:A116 = EIN, 3: BOASG
         $OUT[116] = TRUE
      ;ENDFOLD
      ;FOLD A130 = EIN ;%{SE}%MKUKATPVW %CVW_SPS %VBOASG %P 2:A130 = EIN, 3: BOASG
         $OUT[130] = TRUE
      ;ENDFOLD
      ;FOLD -- Quitt. Fraesen SK1 AUS -- ;%{SE}%MKUKATPVW %CVW_COM %VCOMMENT %P 2:-- Quitt. Fraesen SK1 AUS --, 3: VW_COMMENT
      ;ENDFOLD
      ;FOLD A786 = F830 ;%{SE}%MKUKATPVW %CVW_SPS %VBOASG %P 2:A786 = F830, 3: BOASG
         $OUT[786] = $FLAG[830]
      ;ENDFOLD
      ;FOLD A722 = !F830 ;%{SE}%MKUKATPVW %CVW_SPS %VBOASG %P 2:A722 = !F830, 3: BOASG
         $OUT[722] = NOT $FLAG[830]
      ;ENDFOLD
      ;FOLD Schritt 52 = T8 & A4039  ;%{SE}%MKUKATPVW %CVW_SPS %VST_CON %P 2:Schritt 52 = T8 & A4039 , 3: ST_CON
         IF $TIMER_FLAG[8] AND $OUT[4039] THEN
            PREVSTEP = $APP_INT[5]
            $APP_INT[5] = 52
         ENDIF
      ;ENDFOLD
   ;ENDFOLD
   ;FOLD SCHRITT 52 -- STAT EZ1/SP1/KE1 -- ;%{P}%MKUKATPVW,%CSTEP,%VST_NR,%P 1:SCHRITT, 2:52, 3: STAT EZ1/SP1/KE1
      ;FOLD ;%{H}
         Case 52
      ;ENDFOLD
      ;FOLD -- Hilfsflag SK Programmwechsel -- ;%{SE}%MKUKATPVW %CVW_COM %VCOMMENT %P 2:-- Hilfsflag SK Programmwechsel --, 3: VW_COMMENT
      ;ENDFOLD
      ;FOLD F334 = AUS ;%{SE}%MKUKATPVW %CVW_SPS %VBOASG %P 2:F334 = AUS, 3: BOASG
         $FLAG[334] = FALSE
      ;ENDFOLD
      ;FOLD -- Ueberwachungszeit KF1 EIN -- ;%{SE}%MKUKATPVW %CVW_COM %VCOMMENT %P 2:-- Ueberwachungszeit KF1 EIN --, 3: VW_COMMENT
      ;ENDFOLD
      ;FOLD T7 ( EIN ) = -50[1/10Sek] ;%{SE}%MKUKATPVW %CVW_SPS %VTASG %P 2:T7 ( EIN ) = -50[1/10Sek], 3: TASG
         VW(#SET_TIME,TRUE,7,0,-50)
      ;ENDFOLD
      ;FOLD -- KF1 einschalten -- ;%{SE}%MKUKATPVW %CVW_COM %VCOMMENT %P 2:-- KF1 einschalten --, 3: VW_COMMENT
      ;ENDFOLD
      ;FOLD i1 (EIN) = 0 ;%{SE}%MKUKATPVW %CVW_SPS %VARIASG %P 2:i1 (EIN) = 0, 3: ARIASG
         VW(#COUNTER,TRUE,1,0)
      ;ENDFOLD
      ;FOLD A834 = EIN ;%{SE}%MKUKATPVW %CVW_SPS %VBOASG %P 2:A834 = EIN, 3: BOASG
         $OUT[834] = TRUE
      ;ENDFOLD
      ;FOLD Schritt 53 = A4039  ;%{SE}%MKUKATPVW %CVW_SPS %VST_CON %P 2:Schritt 53 = A4039 , 3: ST_CON
         IF $OUT[4039] THEN
            PREVSTEP = $APP_INT[5]
            $APP_INT[5] = 53
         ENDIF
      ;ENDFOLD
   ;ENDFOLD
   ;FOLD SCHRITT 53 -- STAT EZ1/SP1/KE1 -- ;%{P}%MKUKATPVW,%CSTEP,%VST_NR,%P 1:SCHRITT, 2:53, 3: STAT EZ1/SP1/KE1
      ;FOLD ;%{H}
         Case 53
      ;ENDFOLD
      ;FOLD -- Funktionstest KF Motor -- ;%{SE}%MKUKATPVW %CVW_COM %VCOMMENT %P 2:-- Funktionstest KF Motor --, 3: VW_COMMENT
      ;ENDFOLD
      ;FOLD F312 = EIN ;%{SE}%MKUKATPVW %CVW_SPS %VBOASG %P 2:F312 = EIN, 3: BOASG
         $FLAG[312] = TRUE
      ;ENDFOLD
      ;FOLD F313 = i1 > 2 ;%{SE}%MKUKATPVW %CVW_SPS %VBOCMP %P 2:F313 = i1 > 2, 3: BOCMP
         $FLAG[313] = $COUNT_I[1] > 2
      ;ENDFOLD
      ;FOLD Schritt 54 = (F313 + T7) & A4039  ;%{SE}%MKUKATPVW %CVW_SPS %VST_CON %P 2:Schritt 54 = (F313 + T7) & A4039 , 3: ST_CON
         IF ($FLAG[313] OR $TIMER_FLAG[7]) AND $OUT[4039] THEN
            PREVSTEP = $APP_INT[5]
            $APP_INT[5] = 54
         ENDIF
      ;ENDFOLD
   ;ENDFOLD
   ;FOLD SCHRITT 54 -- STAT EZ1/SP1/KE1-- ;%{P}%MKUKATPVW,%CSTEP,%VST_NR,%P 1:SCHRITT, 2:54, 3: STAT EZ1/SP1/KE1
      ;FOLD ;%{H}
         Case 54
      ;ENDFOLD
      ;FOLD F312 = AUS ;%{SE}%MKUKATPVW %CVW_SPS %VBOASG %P 2:F312 = AUS, 3: BOASG
         $FLAG[312] = FALSE
      ;ENDFOLD
      ;FOLD -- Ueberwachungszeit KS1 schwenken -- ;%{SE}%MKUKATPVW %CVW_COM %VCOMMENT %P 2:-- Ueberwachungszeit KS1 schwenken --, 3: VW_COMMENT
      ;ENDFOLD
      ;FOLD t8 ( EIN ) = -100[1/10Sek] ;%{SE}%MKUKATPVW %CVW_SPS %VTASG %P 2:t8 ( EIN ) = -100[1/10Sek], 3: TASG
         VW(#SET_TIME,TRUE,8,0,-100)
      ;ENDFOLD
      ;FOLD Schritt 55 = A4039  ;%{SE}%MKUKATPVW %CVW_SPS %VST_CON %P 2:Schritt 55 = A4039 , 3: ST_CON
         IF $OUT[4039] THEN
            PREVSTEP = $APP_INT[5]
            $APP_INT[5] = 55
         ENDIF
      ;ENDFOLD
   ;ENDFOLD
   ;FOLD SCHRITT 55 -- STAT EZ1/SP1/KE1 -- ;%{P}%MKUKATPVW,%CSTEP,%VST_NR,%P 1:SCHRITT, 2:55, 3: STAT EZ1/SP1/KE1
      ;FOLD ;%{H}
         Case 55
      ;ENDFOLD
      ;FOLD -- RSK Fehlerausgabe KF1 Initiator/Motor -- ;%{SE}%MKUKATPVW %CVW_COM %VCOMMENT %P 2:-- RSK Fehlerausgabe KF1 Initiator/Motor --, 3: VW_COMMENT
      ;ENDFOLD
      ;FOLD F322 = !F313 ;%{SE}%MKUKATPVW %CVW_SPS %VBOASG %P 2:F322 = !F313, 3: BOASG
         $FLAG[322] = NOT $FLAG[313]
      ;ENDFOLD
      ;FOLD -- RSK Fehlerausgabe KS1 Ruhest. -- ;%{SE}%MKUKATPVW %CVW_COM %VCOMMENT %P 2:-- RSK Fehlerausgabe KS1 Ruhest. --, 3: VW_COMMENT
      ;ENDFOLD
      ;FOLD F323 = (!E842 + E843 + E844 + !E845) & !F324 & !F328 ;%{SE}%MKUKATPVW %CVW_SPS %VBOASG %P 2:F323 = (!E842 + E843 + E844 + !E845) & !F324 & !F328, 3: BOASG
         $FLAG[323] = (NOT $IN[842] OR $IN[843] OR $IN[844] OR NOT $IN[845]) AND NOT $FLAG[324] AND NOT $FLAG[328]
      ;ENDFOLD
      ;FOLD -- RSK Sammelstoerung -- ;%{SE}%MKUKATPVW %CVW_COM %VCOMMENT %P 2:-- RSK Sammelstoerung --, 3: VW_COMMENT
      ;ENDFOLD
      ;FOLD F329 = F322 + F323 + T8 ;%{SE}%MKUKATPVW %CVW_SPS %VBOASG %P 2:F329 = F322 + F323 + T8, 3: BOASG
         $FLAG[329] = $FLAG[322] OR $FLAG[323] OR $TIMER_FLAG[8]
      ;ENDFOLD
      ;FOLD T7 ( EIN ) = STOP ;%{SE}%MKUKATPVW %CVW_SPS %VTSTOP %P 2:T7 ( EIN ) = STOP, 3: TSTOP
         VW(#SET_TIME,TRUE,7,1,0)
      ;ENDFOLD
      ;FOLD A834 = !F322 & !F323 ;%{SE}%MKUKATPVW %CVW_SPS %VBOASG %P 2:A834 = !F322 & !F323, 3: BOASG
         $OUT[834] = NOT $FLAG[322] AND NOT $FLAG[323]
      ;ENDFOLD
      ;FOLD -- KF1 Versetzeinheit vor -- ;%{SE}%MKUKATPVW %CVW_COM %VCOMMENT %P 2:-- KF1 Versetzeinheit vor --, 3: VW_COMMENT
      ;ENDFOLD
      ;FOLD A835 = !F322 & !F323 & F564 ;%{SE}%MKUKATPVW %CVW_SPS %VBOASG %P 2:A835 = !F322 & !F323 & F564, 3: BOASG
         $OUT[835] = NOT $FLAG[322] AND NOT $FLAG[323] AND $FLAG[564]
      ;ENDFOLD
      ;FOLD Schritt 56 = (!F322 & !F323 & (E835 & F564 + !E835 & !F564) + T8) & A4039  ;%{SE}%MKUKATPVW %CVW_SPS %VST_CON %P 2:Schritt 56 = (!F322 & !F323 & (E835 & F564 + !E835 & !F564) + T8) & A4039 , 3: ST_CON
         IF (NOT $FLAG[322] AND NOT $FLAG[323] AND ($IN[835] AND $FLAG[564] OR NOT $IN[835] AND NOT $FLAG[564]) OR $TIMER_FLAG[8]) AND $OUT[4039] THEN
            PREVSTEP = $APP_INT[5]
            $APP_INT[5] = 56
         ENDIF
      ;ENDFOLD
      ;FOLD Schritt 72 = (F322 + F323) & !F324 & !F328 & A4039  ;%{SE}%MKUKATPVW %CVW_SPS %VST_CON %P 2:Schritt 72 = (F322 + F323) & !F324 & !F328 & A4039 , 3: ST_CON
         IF ($FLAG[322] OR $FLAG[323]) AND NOT $FLAG[324] AND NOT $FLAG[328] AND $OUT[4039] THEN
            PREVSTEP = $APP_INT[5]
            $APP_INT[5] = 72
         ENDIF
      ;ENDFOLD
   ;ENDFOLD
   ;FOLD SCHRITT 56 -- STAT EZ1/SP1/KE1 -- ;%{P}%MKUKATPVW,%CSTEP,%VST_NR,%P 1:SCHRITT, 2:56, 3: STAT EZ1/SP1/KE1
      ;FOLD ;%{H}
         Case 56
      ;ENDFOLD
      ;FOLD -- RSK Sammelstoerung -- ;%{SE}%MKUKATPVW %CVW_COM %VCOMMENT %P 2:-- RSK Sammelstoerung --, 3: VW_COMMENT
      ;ENDFOLD
      ;FOLD F329 = T8 ;%{SE}%MKUKATPVW %CVW_SPS %VBOASG %P 2:F329 = T8, 3: BOASG
         $FLAG[329] = $TIMER_FLAG[8]
      ;ENDFOLD
      ;FOLD F324 = AUS ;%{SE}%MKUKATPVW %CVW_SPS %VBOASG %P 2:F324 = AUS, 3: BOASG
         $FLAG[324] = FALSE
      ;ENDFOLD
      ;FOLD F328 = AUS ;%{SE}%MKUKATPVW %CVW_SPS %VBOASG %P 2:F328 = AUS, 3: BOASG
         $FLAG[328] = FALSE
      ;ENDFOLD
      ;FOLD -- KS1 in Arbeitsstellung schwenken -- ;%{SE}%MKUKATPVW %CVW_COM %VCOMMENT %P 2:-- KS1 in Arbeitsstellung schwenken --, 3: VW_COMMENT
      ;ENDFOLD
      ;FOLD A842 = (F745 + !F714) & (E717 + F714) & !E843 & (E835 & F564 + !E835 & !F564) ;%{SE}%MKUKATPVW %CVW_SPS %VBOASG %P 2:A842 = (F745 + !F714) & (E717 + F714) & !E843 & (E835 & F564 + !E835 & !F564), 3: BOASG
         $OUT[842] = ($FLAG[745] OR NOT $FLAG[714]) AND ($IN[717] OR $FLAG[714]) AND NOT $IN[843] AND ($IN[835] AND $FLAG[564] OR NOT $IN[835] AND NOT $FLAG[564])
      ;ENDFOLD
      ;FOLD -- KF1 Ausblasen -- ;%{SE}%MKUKATPVW %CVW_COM %VCOMMENT %P 2:-- KF1 Ausblasen --, 3: VW_COMMENT
      ;ENDFOLD
      ;FOLD A847 = F330 + !F330 & !F331 & !F332 ;%{SE}%MKUKATPVW %CVW_SPS %VBOASG %P 2:A847 = F330 + !F330 & !F331 & !F332, 3: BOASG
         $OUT[847] = $FLAG[330] OR NOT $FLAG[330] AND NOT $FLAG[331] AND NOT $FLAG[332]
      ;ENDFOLD
      ;FOLD Schritt 57 = (F745 + !F714) & (E717 + F714) & (A842 + E843 + T8) & A4039  ;%{SE}%MKUKATPVW %CVW_SPS %VST_CON %P 2:Schritt 57 = (F745 + !F714) & (E717 + F714) & (A842 + E843 + T8) & A4039 , 3: ST_CON
         IF ($FLAG[745] OR NOT $FLAG[714]) AND ($IN[717] OR $FLAG[714]) AND ($OUT[842] OR $IN[843] OR $TIMER_FLAG[8]) AND $OUT[4039] THEN
            PREVSTEP = $APP_INT[5]
            $APP_INT[5] = 57
         ENDIF
      ;ENDFOLD
   ;ENDFOLD
   ;FOLD SCHRITT 57 -- STAT EZ1/SP1/KE1 -- ;%{P}%MKUKATPVW,%CSTEP,%VST_NR,%P 1:SCHRITT, 2:57, 3: STAT EZ1/SP1/KE1
      ;FOLD ;%{H}
         Case 57
      ;ENDFOLD
      ;FOLD -- RSK Fehlerausgabe KF Versetzeinheit -- ;%{SE}%MKUKATPVW %CVW_COM %VCOMMENT %P 2:-- RSK Fehlerausgabe KF Versetzeinheit --, 3: VW_COMMENT
      ;ENDFOLD
      ;FOLD F328 = !E835 & F564 & !F324 ;%{SE}%MKUKATPVW %CVW_SPS %VBOASG %P 2:F328 = !E835 & F564 & !F324, 3: BOASG
         $FLAG[328] = NOT $IN[835] AND $FLAG[564] AND NOT $FLAG[324]
      ;ENDFOLD
      ;FOLD -- RSK Fehlerausgabe KS1 Arbeitsstellung -- ;%{SE}%MKUKATPVW %CVW_COM %VCOMMENT %P 2:-- RSK Fehlerausgabe KS1 Arbeitsstellung --, 3: VW_COMMENT
      ;ENDFOLD
      ;FOLD F324 = (E842 + !E843 + !E844 + E845) & T8 & (E835 + !F564) + F324 ;%{SE}%MKUKATPVW %CVW_SPS %VBOASG %P 2:F324 = (E842 + !E843 + !E844 + E845) & T8 & (E835 + !F564) + F324, 3: BOASG
         $FLAG[324] = ($IN[842] OR NOT $IN[843] OR NOT $IN[844] OR $IN[845]) AND $TIMER_FLAG[8] AND ($IN[835] OR NOT $FLAG[564]) OR $FLAG[324]
      ;ENDFOLD
      ;FOLD -- RSK Fehlerausgabe EZ/SP min. Oeffnung -- ;%{SE}%MKUKATPVW %CVW_COM %VCOMMENT %P 2:-- RSK Fehlerausgabe EZ/SP min. Oeffnung --, 3: VW_COMMENT
      ;ENDFOLD
      ;FOLD F333 = !F745 ;%{SE}%MKUKATPVW %CVW_SPS %VBOASG %P 2:F333 = !F745, 3: BOASG
         $FLAG[333] = NOT $FLAG[745]
      ;ENDFOLD
      ;FOLD -- RSK Sammelstoerung -- ;%{SE}%MKUKATPVW %CVW_COM %VCOMMENT %P 2:-- RSK Sammelstoerung --, 3: VW_COMMENT
      ;ENDFOLD
      ;FOLD F329 = F324 + F328 + F333 ;%{SE}%MKUKATPVW %CVW_SPS %VBOASG %P 2:F329 = F324 + F328 + F333, 3: BOASG
         $FLAG[329] = $FLAG[324] OR $FLAG[328] OR $FLAG[333]
      ;ENDFOLD
      ;FOLD A834 = !F324 & !F328 ;%{SE}%MKUKATPVW %CVW_SPS %VBOASG %P 2:A834 = !F324 & !F328, 3: BOASG
         $OUT[834] = NOT $FLAG[324] AND NOT $FLAG[328]
      ;ENDFOLD
      ;FOLD -- KF1 Ausblasen -- ;%{SE}%MKUKATPVW %CVW_COM %VCOMMENT %P 2:-- KF1 Ausblasen --, 3: VW_COMMENT
      ;ENDFOLD
      ;FOLD A847 = (F330 + !F330 & !F331 & !F332) & !F324 & !F328 ;%{SE}%MKUKATPVW %CVW_SPS %VBOASG %P 2:A847 = (F330 + !F330 & !F331 & !F332) & !F324 & !F328, 3: BOASG
         $OUT[847] = ($FLAG[330] OR NOT $FLAG[330] AND NOT $FLAG[331] AND NOT $FLAG[332]) AND NOT $FLAG[324] AND NOT $FLAG[328]
      ;ENDFOLD
      ;FOLD A835 = F564 ;%{SE}%MKUKATPVW %CVW_SPS %VBOASG %P 2:A835 = F564, 3: BOASG
         $OUT[835] = $FLAG[564]
      ;ENDFOLD
      ;FOLD -- Ueberwachungszeit EZ1/SP1/KE1 SZ1 schliessen -- ;%{SE}%MKUKATPVW %CVW_COM %VCOMMENT %P 2:-- Ueberwachungszeit EZ1/SP1/KE1 SZ1 schliessen --, 3: VW_COMMENT
      ;ENDFOLD
      ;FOLD t9 ( EIN ) = -80[1/10Sek] ;%{SE}%MKUKATPVW %CVW_SPS %VTASG %P 2:t9 ( EIN ) = -80[1/10Sek], 3: TASG
         VW(#SET_TIME,TRUE,9,0,-80)
      ;ENDFOLD
      ;FOLD -- Verweilzeit Versetzeinheit Rueck -- ;%{SE}%MKUKATPVW %CVW_COM %VCOMMENT %P 2:-- Verweilzeit Versetzeinheit Rueck --, 3: VW_COMMENT
      ;ENDFOLD
      ;FOLD t11 ( EIN ) = i24[1/10Sek] ;%{SE}%MKUKATPVW %CVW_SPS %VTASG %P 2:t11 ( EIN ) = i24[1/10Sek], 3: TASG
         VW(#SET_TIME,TRUE,11,0,$COUNT_I[24])
      ;ENDFOLD
      ;FOLD Schritt 52 = (F324 + F328) & (E26 + E27) & A4039  ;%{SE}%MKUKATPVW %CVW_SPS %VST_CON %P 2:Schritt 52 = (F324 + F328) & (E26 + E27) & A4039 , 3: ST_CON
         IF ($FLAG[324] OR $FLAG[328]) AND ($IN[26] OR $IN[27]) AND $OUT[4039] THEN
            PREVSTEP = $APP_INT[5]
            $APP_INT[5] = 52
         ENDIF
      ;ENDFOLD
      ;FOLD Schritt 58 = !F324 & !F328 & !E842 & E843 & E844 & !E845 & A4039  ;%{SE}%MKUKATPVW %CVW_SPS %VST_CON %P 2:Schritt 58 = !F324 & !F328 & !E842 & E843 & E844 & !E845 & A4039 , 3: ST_CON
         IF NOT $FLAG[324] AND NOT $FLAG[328] AND NOT $IN[842] AND $IN[843] AND $IN[844] AND NOT $IN[845] AND $OUT[4039] THEN
            PREVSTEP = $APP_INT[5]
            $APP_INT[5] = 58
         ENDIF
      ;ENDFOLD
   ;ENDFOLD
   ;FOLD SCHRITT 58 -- STAT EZ1/SP1/KE1-- ;%{P}%MKUKATPVW,%CSTEP,%VST_NR,%P 1:SCHRITT, 2:58, 3: STAT EZ1/SP1/KE1
      ;FOLD ;%{H}
         Case 58
      ;ENDFOLD
      ;FOLD -- Umdreh. KF setzen zwischenspeichern -- ;%{SE}%MKUKATPVW %CVW_COM %VCOMMENT %P 2:-- Umdreh. KF setzen zwischenspeichern --, 3: VW_COMMENT
      ;ENDFOLD
      ;FOLD F270 = F99 & F732 ;%{SE}%MKUKATPVW %CVW_SPS %VBOASG %P 2:F270 = F99 & F732, 3: BOASG
         $FLAG[270] = $FLAG[99] AND $FLAG[732]
      ;ENDFOLD
      ;FOLD i45 ( EIN ) = i4 ;%{SE}%MKUKATPVW %CVW_SPS %VARIASG %P 2:i45 ( EIN ) = i4, 3: ARIASG
         VW(#COUNTER,TRUE,45,$COUNT_I[4])
      ;ENDFOLD
      ;FOLD i4 ( F270 ) = i43 ;%{SE}%MKUKATPVW %CVW_SPS %VARIASG %P 2:i4 ( F270 ) = i43, 3: ARIASG
         VW(#COUNTER,$FLAG[270],4,$COUNT_I[43])
      ;ENDFOLD
      ;FOLD i1 ( EIN ) = 0 ;%{SE}%MKUKATPVW %CVW_SPS %VARIASG %P 2:i1 ( EIN ) = 0, 3: ARIASG
         VW(#COUNTER,TRUE,1,0)
      ;ENDFOLD
      ;FOLD F98 = AUS ;%{SE}%MKUKATPVW %CVW_SPS %VBOASG %P 2:F98 = AUS, 3: BOASG
         $FLAG[98] = FALSE
      ;ENDFOLD
      ;FOLD F312 = AUS ;%{SE}%MKUKATPVW %CVW_SPS %VBOASG %P 2:F312 = AUS, 3: BOASG
         $FLAG[312] = FALSE
      ;ENDFOLD
      ;FOLD F313 = AUS ;%{SE}%MKUKATPVW %CVW_SPS %VBOASG %P 2:F313 = AUS, 3: BOASG
         $FLAG[313] = FALSE
      ;ENDFOLD
      ;FOLD F324 = AUS ;%{SE}%MKUKATPVW %CVW_SPS %VBOASG %P 2:F324 = AUS, 3: BOASG
         $FLAG[324] = FALSE
      ;ENDFOLD
      ;FOLD F328 = AUS ;%{SE}%MKUKATPVW %CVW_SPS %VBOASG %P 2:F328 = AUS, 3: BOASG
         $FLAG[328] = FALSE
      ;ENDFOLD
      ;FOLD -- KF1 einschalten nach Fehler -- ;%{SE}%MKUKATPVW %CVW_COM %VCOMMENT %P 2:-- KF1 einschalten nach Fehler --, 3: VW_COMMENT
      ;ENDFOLD
      ;FOLD A834 = EIN ;%{SE}%MKUKATPVW %CVW_SPS %VBOASG %P 2:A834 = EIN, 3: BOASG
         $OUT[834] = TRUE
      ;ENDFOLD
      ;FOLD -- KF1 Versetzeinheit rueck -- ;%{SE}%MKUKATPVW %CVW_COM %VCOMMENT %P 2:-- KF1 Versetzeinheit rueck --, 3: VW_COMMENT
      ;ENDFOLD
      ;FOLD A835 = AUS ;%{SE}%MKUKATPVW %CVW_SPS %VBOASG %P 2:A835 = AUS, 3: BOASG
         $OUT[835] = FALSE
      ;ENDFOLD
      ;FOLD Schritt 59 = T11 & A4039  ;%{SE}%MKUKATPVW %CVW_SPS %VST_CON %P 2:Schritt 59 = T11 & A4039 , 3: ST_CON
         IF $TIMER_FLAG[11] AND $OUT[4039] THEN
            PREVSTEP = $APP_INT[5]
            $APP_INT[5] = 59
         ENDIF
      ;ENDFOLD
   ;ENDFOLD
   ;FOLD SCHRITT 59 -- STAT EZ1/SP1/KE1 -- ;%{P}%MKUKATPVW,%CSTEP,%VST_NR,%P 1:SCHRITT, 2:59, 3: STAT EZ1/SP1/KE1
      ;FOLD ;%{H}
         Case 59
      ;ENDFOLD
      ;FOLD F270 = AUS ;%{SE}%MKUKATPVW %CVW_SPS %VBOASG %P 2:F270 = AUS, 3: BOASG
         $FLAG[270] = FALSE
      ;ENDFOLD
      ;FOLD t11 ( EIN ) = STOP ;%{SE}%MKUKATPVW %CVW_SPS %VTSTOP %P 2:t11 ( EIN ) = STOP, 3: TSTOP
         VW(#SET_TIME,TRUE,11,1,0)
      ;ENDFOLD
      ;FOLD -- EZ1/SP1/KE1 SZ1 schliessen -- ;%{SE}%MKUKATPVW %CVW_COM %VCOMMENT %P 2:-- EZ1/SP1/KE1 SZ1 schliessen --, 3: VW_COMMENT
      ;ENDFOLD
      ;FOLD A717 = AUS ;%{SE}%MKUKATPVW %CVW_SPS %VBOASG %P 2:A717 = AUS, 3: BOASG
         $OUT[717] = FALSE
      ;ENDFOLD
      ;FOLD A718 = EIN ;%{SE}%MKUKATPVW %CVW_SPS %VBOASG %P 2:A718 = EIN, 3: BOASG
         $OUT[718] = TRUE
      ;ENDFOLD
      ;FOLD -- KF1 Ausblasen -- ;%{SE}%MKUKATPVW %CVW_COM %VCOMMENT %P 2:-- KF1 Ausblasen --, 3: VW_COMMENT
      ;ENDFOLD
      ;FOLD A847 = F330 + F331 + !F330 & !F331 & !F332 ;%{SE}%MKUKATPVW %CVW_SPS %VBOASG %P 2:A847 = F330 + F331 + !F330 & !F331 & !F332, 3: BOASG
         $OUT[847] = $FLAG[330] OR $FLAG[331] OR NOT $FLAG[330] AND NOT $FLAG[331] AND NOT $FLAG[332]
      ;ENDFOLD
      ;FOLD Schritt 60 = (!E717 & E718 + T9) & A4039  ;%{SE}%MKUKATPVW %CVW_SPS %VST_CON %P 2:Schritt 60 = (!E717 & E718 + T9) & A4039 , 3: ST_CON
         IF (NOT $IN[717] AND $IN[718] OR $TIMER_FLAG[9]) AND $OUT[4039] THEN
            PREVSTEP = $APP_INT[5]
            $APP_INT[5] = 60
         ENDIF
      ;ENDFOLD
   ;ENDFOLD
   ;FOLD SCHRITT 60 -- STAT EZ1/SP1/KE1 -- ;%{P}%MKUKATPVW,%CSTEP,%VST_NR,%P 1:SCHRITT, 2:60, 3: STAT EZ1/SP1/KE1
      ;FOLD ;%{H}
         Case 60
      ;ENDFOLD
      ;FOLD -- RSK Fehlerausgabe Kraftaufbau -- ;%{SE}%MKUKATPVW %CVW_COM %VCOMMENT %P 2:-- RSK Fehlerausgabe Kraftaufbau --, 3: VW_COMMENT
      ;ENDFOLD
      ;FOLD F325 = T9 ;%{SE}%MKUKATPVW %CVW_SPS %VBOASG %P 2:F325 = T9, 3: BOASG
         $FLAG[325] = $TIMER_FLAG[9]
      ;ENDFOLD
      ;FOLD -- RSK Sammelstoerung -- ;%{SE}%MKUKATPVW %CVW_COM %VCOMMENT %P 2:-- RSK Sammelstoerung --, 3: VW_COMMENT
      ;ENDFOLD
      ;FOLD F329 = F325 ;%{SE}%MKUKATPVW %CVW_SPS %VBOASG %P 2:F329 = F325, 3: BOASG
         $FLAG[329] = $FLAG[325]
      ;ENDFOLD
      ;FOLD -- KF1 abschalten bei Fehler -- ;%{SE}%MKUKATPVW %CVW_COM %VCOMMENT %P 2:-- KF1 abschalten bei Fehler --, 3: VW_COMMENT
      ;ENDFOLD
      ;FOLD A834 = !T9 ;%{SE}%MKUKATPVW %CVW_SPS %VBOASG %P 2:A834 = !T9, 3: BOASG
         $OUT[834] = NOT $TIMER_FLAG[9]
      ;ENDFOLD
      ;FOLD -- KF1 Ausblasen -- ;%{SE}%MKUKATPVW %CVW_COM %VCOMMENT %P 2:-- KF1 Ausblasen --, 3: VW_COMMENT
      ;ENDFOLD
      ;FOLD A847 = (F330 + F331 + !F330 & !F331 & !F332) & !T9 ;%{SE}%MKUKATPVW %CVW_SPS %VBOASG %P 2:A847 = (F330 + F331 + !F330 & !F331 & !F332) & !T9, 3: BOASG
         $OUT[847] = ($FLAG[330] OR $FLAG[331] OR NOT $FLAG[330] AND NOT $FLAG[331] AND NOT $FLAG[332]) AND NOT $TIMER_FLAG[9]
      ;ENDFOLD
      ;FOLD -- Warte Fraesen fertig oder Timeout -- ;%{SE}%MKUKATPVW %CVW_COM %VCOMMENT %P 2:-- Warte Fraesen fertig oder Timeout --, 3: VW_COMMENT
      ;ENDFOLD
      ;FOLD Schritt 61 = (F79 & F98 + F78 & F94 & !F287 + T7 + T9 + F325) & A4039  ;%{SE}%MKUKATPVW %CVW_SPS %VST_CON %P 2:Schritt 61 = (F79 & F98 + F78 & F94 & !F287 + T7 + T9 + F325) & A4039 , 3: ST_CON
         IF ($FLAG[79] AND $FLAG[98] OR $FLAG[78] AND $FLAG[94] AND NOT $FLAG[287] OR $TIMER_FLAG[7] OR $TIMER_FLAG[9] OR $FLAG[325]) AND $OUT[4039] THEN
            PREVSTEP = $APP_INT[5]
            $APP_INT[5] = 61
         ENDIF
      ;ENDFOLD
      ;FOLD Schritt 61 = (F78 & F96 & F287 + T7 + T9 + F325) & A4039  ;%{SE}%MKUKATPVW %CVW_SPS %VST_CON %P 2:Schritt 61 = (F78 & F96 & F287 + T7 + T9 + F325) & A4039 , 3: ST_CON
         IF ($FLAG[78] AND $FLAG[96] AND $FLAG[287] OR $TIMER_FLAG[7] OR $TIMER_FLAG[9] OR $FLAG[325]) AND $OUT[4039] THEN
            PREVSTEP = $APP_INT[5]
            $APP_INT[5] = 61
         ENDIF
      ;ENDFOLD
   ;ENDFOLD
   ;FOLD SCHRITT 61 -- STAT EZ1/SP1/KE1-- ;%{P}%MKUKATPVW,%CSTEP,%VST_NR,%P 1:SCHRITT, 2:61, 3: STAT EZ1/SP1/KE1
      ;FOLD ;%{H}
         Case 61
      ;ENDFOLD
      ;FOLD -- EZ1/SP1/KE1 SZ1 oeffnen -- ;%{SE}%MKUKATPVW %CVW_COM %VCOMMENT %P 2:-- EZ1/SP1/KE1 SZ1 oeffnen --, 3: VW_COMMENT
      ;ENDFOLD
      ;FOLD t9 ( EIN ) = STOP ;%{SE}%MKUKATPVW %CVW_SPS %VTSTOP %P 2:t9 ( EIN ) = STOP, 3: TSTOP
         VW(#SET_TIME,TRUE,9,1,0)
      ;ENDFOLD
      ;FOLD A719 = AUS ;%{SE}%MKUKATPVW %CVW_SPS %VBOASG %P 2:A719 = AUS, 3: BOASG
         $OUT[719] = FALSE
      ;ENDFOLD
      ;FOLD A718 = AUS ;%{SE}%MKUKATPVW %CVW_SPS %VBOASG %P 2:A718 = AUS, 3: BOASG
         $OUT[718] = FALSE
      ;ENDFOLD
      ;FOLD A717 = EIN ;%{SE}%MKUKATPVW %CVW_SPS %VBOASG %P 2:A717 = EIN, 3: BOASG
         $OUT[717] = TRUE
      ;ENDFOLD
      ;FOLD -- KF1 Ausblasen -- ;%{SE}%MKUKATPVW %CVW_COM %VCOMMENT %P 2:-- KF1 Ausblasen --, 3: VW_COMMENT
      ;ENDFOLD
      ;FOLD A847 = (F330 + F331 + F332 + !F330 & !F331 & !F332) & !T9 ;%{SE}%MKUKATPVW %CVW_SPS %VBOASG %P 2:A847 = (F330 + F331 + F332 + !F330 & !F331 & !F332) & !T9, 3: BOASG
         $OUT[847] = ($FLAG[330] OR $FLAG[331] OR $FLAG[332] OR NOT $FLAG[330] AND NOT $FLAG[331] AND NOT $FLAG[332]) AND NOT $TIMER_FLAG[9]
      ;ENDFOLD
      ;FOLD -- KF Ausblasen Ausschaltverzoegerung starten -- ;%{SE}%MKUKATPVW %CVW_COM %VCOMMENT %P 2:-- KF Ausblasen Ausschaltverzoegerung starten --, 3: VW_COMMENT
      ;ENDFOLD
      ;FOLD F737 = EIN ;%{SE}%MKUKATPVW %CVW_SPS %VBOASG %P 2:F737 = EIN, 3: BOASG
         $FLAG[737] = TRUE
      ;ENDFOLD
      ;FOLD -- RSK Sammelstoerung -- ;%{SE}%MKUKATPVW %CVW_COM %VCOMMENT %P 2:-- RSK Sammelstoerung --, 3: VW_COMMENT
      ;ENDFOLD
      ;FOLD F329 = T7 + T9 + F325 ;%{SE}%MKUKATPVW %CVW_SPS %VBOASG %P 2:F329 = T7 + T9 + F325, 3: BOASG
         $FLAG[329] = $TIMER_FLAG[7] OR $TIMER_FLAG[9] OR $FLAG[325]
      ;ENDFOLD
      ;FOLD -- Hilfsflag Startfraesen -- ;%{SE}%MKUKATPVW %CVW_COM %VCOMMENT %P 2:-- Hilfsflag Startfraesen --, 3: VW_COMMENT
      ;ENDFOLD
      ;FOLD F96 = F96 & F287 ;%{SE}%MKUKATPVW %CVW_SPS %VBOASG %P 2:F96 = F96 & F287, 3: BOASG
         $FLAG[96] = $FLAG[96] AND $FLAG[287]
      ;ENDFOLD
      ;FOLD F96 = (F96 & F78 + F98 & F79) & F287 ;%{SE}%MKUKATPVW %CVW_SPS %VBOASG %P 2:F96 = (F96 & F78 + F98 & F79) & F287, 3: BOASG
         $FLAG[96] = ($FLAG[96] AND $FLAG[78] OR $FLAG[98] AND $FLAG[79]) AND $FLAG[287]
      ;ENDFOLD
      ;FOLD F98 = !F130 & F98 + F130 & F287 & F98 ;%{SE}%MKUKATPVW %CVW_SPS %VBOASG %P 2:F98 = !F130 & F98 + F130 & F287 & F98, 3: BOASG
         $FLAG[98] = NOT $FLAG[130] AND $FLAG[98] OR $FLAG[130] AND $FLAG[287] AND $FLAG[98]
      ;ENDFOLD
      ;FOLD F287 = F78 + F79 & F130 ;%{SE}%MKUKATPVW %CVW_SPS %VBOASG %P 2:F287 = F78 + F79 & F130, 3: BOASG
         $FLAG[287] = $FLAG[78] OR $FLAG[79] AND $FLAG[130]
      ;ENDFOLD
      ;FOLD -- Neues Fraesprogramm und Zaehler ruecksetzen -- ;%{SE}%MKUKATPVW %CVW_COM %VCOMMENT %P 2:-- Neues Fraesprogramm und Zaehler ruecksetzen --, 3: VW_COMMENT
      ;ENDFOLD
      ;FOLD F270 = F96 & F732 ;%{SE}%MKUKATPVW %CVW_SPS %VBOASG %P 2:F270 = F96 & F732, 3: BOASG
         $FLAG[270] = $FLAG[96] AND $FLAG[732]
      ;ENDFOLD
      ;FOLD bin3 ( F732 ) = 36 ;%{SE}%MKUKATPVW %CVW_SPS %VARIASG %P 2:bin3 ( F732 ) = 36, 3: ARIASG
         VW(#BINOUT,$FLAG[732],3,36)
      ;ENDFOLD
      ;FOLD i4 ( F270 ) = i45 ;%{SE}%MKUKATPVW %CVW_SPS %VARIASG %P 2:i4 ( F270 ) = i45, 3: ARIASG
         VW(#COUNTER,$FLAG[270],4,$COUNT_I[45])
      ;ENDFOLD
      ;FOLD -- Wiederholung beim Startfraesen -- ;%{SE}%MKUKATPVW %CVW_COM %VCOMMENT %P 2:-- Wiederholung beim Startfraesen --, 3: VW_COMMENT
      ;ENDFOLD
      ;FOLD Schritt 58 = E717 & !E718 & (F78 & !F96 + F79 & F130 & !F96) & !F329 & A4039  ;%{SE}%MKUKATPVW %CVW_SPS %VST_CON %P 2:Schritt 58 = E717 & !E718 & (F78 & !F96 + F79 & F130 & !F96) & !F329 & A4039 , 3: ST_CON
         IF $IN[717] AND NOT $IN[718] AND ($FLAG[78] AND NOT $FLAG[96] OR $FLAG[79] AND $FLAG[130] AND NOT $FLAG[96]) AND NOT $FLAG[329] AND $OUT[4039] THEN
            PREVSTEP = $APP_INT[5]
            $APP_INT[5] = 58
         ENDIF
      ;ENDFOLD
      ;FOLD -- Weiter wenn Fraesen fertig -- ;%{SE}%MKUKATPVW %CVW_COM %VCOMMENT %P 2:-- Weiter wenn Fraesen fertig --, 3: VW_COMMENT
      ;ENDFOLD
      ;FOLD Schritt 62 = E717 & !E718 & (F79 & F98 & (!F130 + F96) + F78 & F96 + F329 + F325) & A4039  ;%{SE}%MKUKATPVW %CVW_SPS %VST_CON %P 2:Schritt 62 = E717 & !E718 & (F79 & F98 & (!F130 + F96) + F78 & F96 + F329 + F325) & A4039 , 3: ST_CON
         IF $IN[717] AND NOT $IN[718] AND ($FLAG[79] AND $FLAG[98] AND (NOT $FLAG[130] OR $FLAG[96]) OR $FLAG[78] AND $FLAG[96] OR $FLAG[329] OR $FLAG[325]) AND $OUT[4039] THEN
            PREVSTEP = $APP_INT[5]
            $APP_INT[5] = 62
         ENDIF
      ;ENDFOLD
   ;ENDFOLD
   ;FOLD SCHRITT 62 -- STAT EZ1/SP1/KE1-- ;%{P}%MKUKATPVW,%CSTEP,%VST_NR,%P 1:SCHRITT, 2:62, 3: STAT EZ1/SP1/KE1
      ;FOLD ;%{H}
         Case 62
      ;ENDFOLD
      ;FOLD F270 = AUS ;%{SE}%MKUKATPVW %CVW_SPS %VBOASG %P 2:F270 = AUS, 3: BOASG
         $FLAG[270] = FALSE
      ;ENDFOLD
      ;FOLD F324 = AUS ;%{SE}%MKUKATPVW %CVW_SPS %VBOASG %P 2:F324 = AUS, 3: BOASG
         $FLAG[324] = FALSE
      ;ENDFOLD
      ;FOLD A717 = AUS ;%{SE}%MKUKATPVW %CVW_SPS %VBOASG %P 2:A717 = AUS, 3: BOASG
         $OUT[717] = FALSE
      ;ENDFOLD
      ;FOLD -- KF1 abschalten -- ;%{SE}%MKUKATPVW %CVW_COM %VCOMMENT %P 2:-- KF1 abschalten --, 3: VW_COMMENT
      ;ENDFOLD
      ;FOLD A834 = AUS ;%{SE}%MKUKATPVW %CVW_SPS %VBOASG %P 2:A834 = AUS, 3: BOASG
         $OUT[834] = FALSE
      ;ENDFOLD
      ;FOLD -- Ueberwachungszeit KF1 Versetzeinheit -- ;%{SE}%MKUKATPVW %CVW_COM %VCOMMENT %P 2:-- Ueberwachungszeit KF1 Versetzeinheit --, 3: VW_COMMENT
      ;ENDFOLD
      ;FOLD t8 ( EIN ) = -40[1/10Sek] ;%{SE}%MKUKATPVW %CVW_SPS %VTASG %P 2:t8 ( EIN ) = -40[1/10Sek], 3: TASG
         VW(#SET_TIME,TRUE,8,0,-40)
      ;ENDFOLD
      ;FOLD Schritt 63 = A4039  ;%{SE}%MKUKATPVW %CVW_SPS %VST_CON %P 2:Schritt 63 = A4039 , 3: ST_CON
         IF $OUT[4039] THEN
            PREVSTEP = $APP_INT[5]
            $APP_INT[5] = 63
         ENDIF
      ;ENDFOLD
   ;ENDFOLD
   ;FOLD SCHRITT 63 -- STAT EZ1/SP1/KE1 -- ;%{P}%MKUKATPVW,%CSTEP,%VST_NR,%P 1:SCHRITT, 2:63, 3: STAT EZ1/SP1/KE1
      ;FOLD ;%{H}
         Case 63
      ;ENDFOLD
      ;FOLD F328 = AUS ;%{SE}%MKUKATPVW %CVW_SPS %VBOASG %P 2:F328 = AUS, 3: BOASG
         $FLAG[328] = FALSE
      ;ENDFOLD
      ;FOLD -- KF1 Versetzeinheit vor -- ;%{SE}%MKUKATPVW %CVW_COM %VCOMMENT %P 2:-- KF1 Versetzeinheit vor --, 3: VW_COMMENT
      ;ENDFOLD
      ;FOLD A835 = F564 ;%{SE}%MKUKATPVW %CVW_SPS %VBOASG %P 2:A835 = F564, 3: BOASG
         $OUT[835] = $FLAG[564]
      ;ENDFOLD
      ;FOLD -- RSK Fehlerausgabe KS1 Arbeitsst. -- ;%{SE}%MKUKATPVW %CVW_COM %VCOMMENT %P 2:-- RSK Fehlerausgabe KS1 Arbeitsst. --, 3: VW_COMMENT
      ;ENDFOLD
      ;FOLD F324 = (E842 + !E843 + !E844 + E845) & !F323 & !F328 + F324 ;%{SE}%MKUKATPVW %CVW_SPS %VBOASG %P 2:F324 = (E842 + !E843 + !E844 + E845) & !F323 & !F328 + F324, 3: BOASG
         $FLAG[324] = ($IN[842] OR NOT $IN[843] OR NOT $IN[844] OR $IN[845]) AND NOT $FLAG[323] AND NOT $FLAG[328] OR $FLAG[324]
      ;ENDFOLD
      ;FOLD -- RSK Sammelstoerung -- ;%{SE}%MKUKATPVW %CVW_COM %VCOMMENT %P 2:-- RSK Sammelstoerung --, 3: VW_COMMENT
      ;ENDFOLD
      ;FOLD F329 = F324 + F325 ;%{SE}%MKUKATPVW %CVW_SPS %VBOASG %P 2:F329 = F324 + F325, 3: BOASG
         $FLAG[329] = $FLAG[324] OR $FLAG[325]
      ;ENDFOLD
      ;FOLD -- Ueberwachungszeit KS1 schwenken -- ;%{SE}%MKUKATPVW %CVW_COM %VCOMMENT %P 2:-- Ueberwachungszeit KS1 schwenken --, 3: VW_COMMENT
      ;ENDFOLD
      ;FOLD t9 ( EIN ) = -100[1/10Sek] ;%{SE}%MKUKATPVW %CVW_SPS %VTASG %P 2:t9 ( EIN ) = -100[1/10Sek], 3: TASG
         VW(#SET_TIME,TRUE,9,0,-100)
      ;ENDFOLD
      ;FOLD Schritt 62 = F324 & (E26 + E27) & A4039  ;%{SE}%MKUKATPVW %CVW_SPS %VST_CON %P 2:Schritt 62 = F324 & (E26 + E27) & A4039 , 3: ST_CON
         IF $FLAG[324] AND ($IN[26] OR $IN[27]) AND $OUT[4039] THEN
            PREVSTEP = $APP_INT[5]
            $APP_INT[5] = 62
         ENDIF
      ;ENDFOLD
      ;FOLD Schritt 64 = (!F324 & (E835 & F564 + !E835 & !F564) + T8 + F325) & A4039  ;%{SE}%MKUKATPVW %CVW_SPS %VST_CON %P 2:Schritt 64 = (!F324 & (E835 & F564 + !E835 & !F564) + T8 + F325) & A4039 , 3: ST_CON
         IF (NOT $FLAG[324] AND ($IN[835] AND $FLAG[564] OR NOT $IN[835] AND NOT $FLAG[564]) OR $TIMER_FLAG[8] OR $FLAG[325]) AND $OUT[4039] THEN
            PREVSTEP = $APP_INT[5]
            $APP_INT[5] = 64
         ENDIF
      ;ENDFOLD
   ;ENDFOLD
   ;FOLD SCHRITT 64 -- STAT EZ1/SP1/KE1-- ;%{P}%MKUKATPVW,%CSTEP,%VST_NR,%P 1:SCHRITT, 2:64, 3: STAT EZ1/SP1/KE1
      ;FOLD ;%{H}
         Case 64
      ;ENDFOLD
      ;FOLD F323 = AUS ;%{SE}%MKUKATPVW %CVW_SPS %VBOASG %P 2:F323 = AUS, 3: BOASG
         $FLAG[323] = FALSE
      ;ENDFOLD
      ;FOLD F328 = AUS ;%{SE}%MKUKATPVW %CVW_SPS %VBOASG %P 2:F328 = AUS, 3: BOASG
         $FLAG[328] = FALSE
      ;ENDFOLD
      ;FOLD -- RSK Sammelstoerung -- ;%{SE}%MKUKATPVW %CVW_COM %VCOMMENT %P 2:-- RSK Sammelstoerung --, 3: VW_COMMENT
      ;ENDFOLD
      ;FOLD F329 = F325 ;%{SE}%MKUKATPVW %CVW_SPS %VBOASG %P 2:F329 = F325, 3: BOASG
         $FLAG[329] = $FLAG[325]
      ;ENDFOLD
      ;FOLD -- KF1 ein -- ;%{SE}%MKUKATPVW %CVW_COM %VCOMMENT %P 2:-- KF1 ein --, 3: VW_COMMENT
      ;ENDFOLD
      ;FOLD A834 = EIN ;%{SE}%MKUKATPVW %CVW_SPS %VBOASG %P 2:A834 = EIN, 3: BOASG
         $OUT[834] = TRUE
      ;ENDFOLD
      ;FOLD -- KS1 in Ruhestellung schwenken -- ;%{SE}%MKUKATPVW %CVW_COM %VCOMMENT %P 2:-- KS1 in Ruhestellung schwenken --, 3: VW_COMMENT
      ;ENDFOLD
      ;FOLD A842 = (F745 + !F714) & (E717 + F714) & (E835 & F564 + !E835 & !F564) ;%{SE}%MKUKATPVW %CVW_SPS %VBOASG %P 2:A842 = (F745 + !F714) & (E717 + F714) & (E835 & F564 + !E835 & !F564), 3: BOASG
         $OUT[842] = ($FLAG[745] OR NOT $FLAG[714]) AND ($IN[717] OR $FLAG[714]) AND ($IN[835] AND $FLAG[564] OR NOT $IN[835] AND NOT $FLAG[564])
      ;ENDFOLD
      ;FOLD Schritt 65 = (F745 + !F714 + T9) & (A842 + T9) & (E717 + F714) & A4039  ;%{SE}%MKUKATPVW %CVW_SPS %VST_CON %P 2:Schritt 65 = (F745 + !F714 + T9) & (A842 + T9) & (E717 + F714) & A4039 , 3: ST_CON
         IF ($FLAG[745] OR NOT $FLAG[714] OR $TIMER_FLAG[9]) AND ($OUT[842] OR $TIMER_FLAG[9]) AND ($IN[717] OR $FLAG[714]) AND $OUT[4039] THEN
            PREVSTEP = $APP_INT[5]
            $APP_INT[5] = 65
         ENDIF
      ;ENDFOLD
   ;ENDFOLD
   ;FOLD SCHRITT 65 -- STAT EZ1/SP1/KE1 -- ;%{P}%MKUKATPVW,%CSTEP,%VST_NR,%P 1:SCHRITT, 2:65, 3: STAT EZ1/SP1/KE1
      ;FOLD ;%{H}
         Case 65
      ;ENDFOLD
      ;FOLD -- Hilfsflag SK Programmwechsel -- ;%{SE}%MKUKATPVW %CVW_COM %VCOMMENT %P 2:-- Hilfsflag SK Programmwechsel --, 3: VW_COMMENT
      ;ENDFOLD
      ;FOLD F334 = AUS ;%{SE}%MKUKATPVW %CVW_SPS %VBOASG %P 2:F334 = AUS, 3: BOASG
         $FLAG[334] = FALSE
      ;ENDFOLD
      ;FOLD -- RSK Fehlerausgabe KF Versetzeinheit -- ;%{SE}%MKUKATPVW %CVW_COM %VCOMMENT %P 2:-- RSK Fehlerausgabe KF Versetzeinheit --, 3: VW_COMMENT
      ;ENDFOLD
      ;FOLD F328 = !E835 & F564 & !F323 + F328 ;%{SE}%MKUKATPVW %CVW_SPS %VBOASG %P 2:F328 = !E835 & F564 & !F323 + F328, 3: BOASG
         $FLAG[328] = NOT $IN[835] AND $FLAG[564] AND NOT $FLAG[323] OR $FLAG[328]
      ;ENDFOLD
      ;FOLD -- RSK Fehlerausgabe KS1 Ruhestellung -- ;%{SE}%MKUKATPVW %CVW_COM %VCOMMENT %P 2:-- RSK Fehlerausgabe KS1 Ruhestellung --, 3: VW_COMMENT
      ;ENDFOLD
      ;FOLD F323 = (!E842 + E843 + E844 + !E845) & T9 & (E835 + !F564) + F323 ;%{SE}%MKUKATPVW %CVW_SPS %VBOASG %P 2:F323 = (!E842 + E843 + E844 + !E845) & T9 & (E835 + !F564) + F323, 3: BOASG
         $FLAG[323] = (NOT $IN[842] OR $IN[843] OR $IN[844] OR NOT $IN[845]) AND $TIMER_FLAG[9] AND ($IN[835] OR NOT $FLAG[564]) OR $FLAG[323]
      ;ENDFOLD
      ;FOLD -- RSK Fehlerausgabe EZ/SP min. Oeffnung -- ;%{SE}%MKUKATPVW %CVW_COM %VCOMMENT %P 2:-- RSK Fehlerausgabe EZ/SP min. Oeffnung --, 3: VW_COMMENT
      ;ENDFOLD
      ;FOLD F333 = !F745 ;%{SE}%MKUKATPVW %CVW_SPS %VBOASG %P 2:F333 = !F745, 3: BOASG
         $FLAG[333] = NOT $FLAG[745]
      ;ENDFOLD
      ;FOLD -- RSK Sammelstoerung -- ;%{SE}%MKUKATPVW %CVW_COM %VCOMMENT %P 2:-- RSK Sammelstoerung --, 3: VW_COMMENT
      ;ENDFOLD
      ;FOLD F329 = F323 + F325 + F328 + F333 ;%{SE}%MKUKATPVW %CVW_SPS %VBOASG %P 2:F329 = F323 + F325 + F328 + F333, 3: BOASG
         $FLAG[329] = $FLAG[323] OR $FLAG[325] OR $FLAG[328] OR $FLAG[333]
      ;ENDFOLD
      ;FOLD A834 = !F323 & !F328 ;%{SE}%MKUKATPVW %CVW_SPS %VBOASG %P 2:A834 = !F323 & !F328, 3: BOASG
         $OUT[834] = NOT $FLAG[323] AND NOT $FLAG[328]
      ;ENDFOLD
      ;FOLD A835 = F564 ;%{SE}%MKUKATPVW %CVW_SPS %VBOASG %P 2:A835 = F564, 3: BOASG
         $OUT[835] = $FLAG[564]
      ;ENDFOLD
      ;FOLD Schritt 63 = (F323 + F328) & (E26 + E27) & A4039  ;%{SE}%MKUKATPVW %CVW_SPS %VST_CON %P 2:Schritt 63 = (F323 + F328) & (E26 + E27) & A4039 , 3: ST_CON
         IF ($FLAG[323] OR $FLAG[328]) AND ($IN[26] OR $IN[27]) AND $OUT[4039] THEN
            PREVSTEP = $APP_INT[5]
            $APP_INT[5] = 63
         ENDIF
      ;ENDFOLD
      ;FOLD Schritt 66 = !A842 & E842 & !E843 & !E844 & E845 & A4039  ;%{SE}%MKUKATPVW %CVW_SPS %VST_CON %P 2:Schritt 66 = !A842 & E842 & !E843 & !E844 & E845 & A4039 , 3: ST_CON
         IF NOT $OUT[842] AND $IN[842] AND NOT $IN[843] AND NOT $IN[844] AND $IN[845] AND $OUT[4039] THEN
            PREVSTEP = $APP_INT[5]
            $APP_INT[5] = 66
         ENDIF
      ;ENDFOLD
   ;ENDFOLD
   ;FOLD SCHRITT 66 -- STAT EZ1/SP1/KE1 -- ;%{P}%MKUKATPVW,%CSTEP,%VST_NR,%P 1:SCHRITT, 2:66, 3: STAT EZ1/SP1/KE1
      ;FOLD ;%{H}
         Case 66
      ;ENDFOLD
      ;FOLD F323 = AUS ;%{SE}%MKUKATPVW %CVW_SPS %VBOASG %P 2:F323 = AUS, 3: BOASG
         $FLAG[323] = FALSE
      ;ENDFOLD
      ;FOLD F328 = AUS ;%{SE}%MKUKATPVW %CVW_SPS %VBOASG %P 2:F328 = AUS, 3: BOASG
         $FLAG[328] = FALSE
      ;ENDFOLD
      ;FOLD -- RSK Sammelstoerung -- ;%{SE}%MKUKATPVW %CVW_COM %VCOMMENT %P 2:-- RSK Sammelstoerung --, 3: VW_COMMENT
      ;ENDFOLD
      ;FOLD F329 = F325 ;%{SE}%MKUKATPVW %CVW_SPS %VBOASG %P 2:F329 = F325, 3: BOASG
         $FLAG[329] = $FLAG[325]
      ;ENDFOLD
      ;FOLD t9 ( EIN ) = STOP ;%{SE}%MKUKATPVW %CVW_SPS %VTSTOP %P 2:t9 ( EIN ) = STOP, 3: TSTOP
         VW(#SET_TIME,TRUE,9,1,0)
      ;ENDFOLD
      ;FOLD -- KF1 Versetzeinheit rueck -- ;%{SE}%MKUKATPVW %CVW_COM %VCOMMENT %P 2:-- KF1 Versetzeinheit rueck --, 3: VW_COMMENT
      ;ENDFOLD
      ;FOLD A835 = AUS ;%{SE}%MKUKATPVW %CVW_SPS %VBOASG %P 2:A835 = AUS, 3: BOASG
         $OUT[835] = FALSE
      ;ENDFOLD
      ;FOLD -- KF1 aus -- ;%{SE}%MKUKATPVW %CVW_COM %VCOMMENT %P 2:-- KF1 aus --, 3: VW_COMMENT
      ;ENDFOLD
      ;FOLD A834 = AUS ;%{SE}%MKUKATPVW %CVW_SPS %VBOASG %P 2:A834 = AUS, 3: BOASG
         $OUT[834] = FALSE
      ;ENDFOLD
      ;FOLD -- KF1 Ausblasen -- ;%{SE}%MKUKATPVW %CVW_COM %VCOMMENT %P 2:-- KF1 Ausblasen --, 3: VW_COMMENT
      ;ENDFOLD
      ;FOLD A847 = (F330 + F331 + F332) & F737 ;%{SE}%MKUKATPVW %CVW_SPS %VBOASG %P 2:A847 = (F330 + F331 + F332) & F737, 3: BOASG
         $OUT[847] = ($FLAG[330] OR $FLAG[331] OR $FLAG[332]) AND $FLAG[737]
      ;ENDFOLD
      ;FOLD bin1 ( !F329 ) = 1 ;%{SE}%MKUKATPVW %CVW_SPS %VARIASG %P 2:bin1 ( !F329 ) = 1, 3: ARIASG
         VW(#BINOUT,NOT $FLAG[329],1,1)
      ;ENDFOLD
      ;FOLD bin3 ( !F329 ) = 1 ;%{SE}%MKUKATPVW %CVW_SPS %VARIASG %P 2:bin3 ( !F329 ) = 1, 3: ARIASG
         VW(#BINOUT,NOT $FLAG[329],3,1)
      ;ENDFOLD
      ;FOLD -- Wartezeit Programmwechsel SK -- ;%{SE}%MKUKATPVW %CVW_COM %VCOMMENT %P 2:-- Wartezeit Programmwechsel SK --, 3: VW_COMMENT
      ;ENDFOLD
      ;FOLD T8 ( !F334 ) = -2[1/10Sek] ;%{SE}%MKUKATPVW %CVW_SPS %VTASG %P 2:T8 ( !F334 ) = -2[1/10Sek], 3: TASG
         VW(#SET_TIME,NOT $FLAG[334],8,0,-2)
      ;ENDFOLD
      ;FOLD -- Hilfsflag SK Programmwechsel -- ;%{SE}%MKUKATPVW %CVW_COM %VCOMMENT %P 2:-- Hilfsflag SK Programmwechsel --, 3: VW_COMMENT
      ;ENDFOLD
      ;FOLD F334 = EIN ;%{SE}%MKUKATPVW %CVW_SPS %VBOASG %P 2:F334 = EIN, 3: BOASG
         $FLAG[334] = TRUE
      ;ENDFOLD
      ;FOLD -- Ueberwachungszeit EZ1/SP1/KE1 SZ1 Messen -- ;%{SE}%MKUKATPVW %CVW_COM %VCOMMENT %P 2:-- Ueberwachungszeit EZ1/SP1/KE1 SZ1 Messen --, 3: VW_COMMENT
      ;ENDFOLD
      ;FOLD t9 ( EIN ) = -150[1/10Sek] ;%{SE}%MKUKATPVW %CVW_SPS %VTASG %P 2:t9 ( EIN ) = -150[1/10Sek], 3: TASG
         VW(#SET_TIME,TRUE,9,0,-150)
      ;ENDFOLD
      ;FOLD Schritt 51 = (F325 + F329) & (E26 + E27) & A4039  ;%{SE}%MKUKATPVW %CVW_SPS %VST_CON %P 2:Schritt 51 = (F325 + F329) & (E26 + E27) & A4039 , 3: ST_CON
         IF ($FLAG[325] OR $FLAG[329]) AND ($IN[26] OR $IN[27]) AND $OUT[4039] THEN
            PREVSTEP = $APP_INT[5]
            $APP_INT[5] = 51
         ENDIF
      ;ENDFOLD
      ;FOLD Schritt 67 = T8 & !F325 & !F329 & A4039  ;%{SE}%MKUKATPVW %CVW_SPS %VST_CON %P 2:Schritt 67 = T8 & !F325 & !F329 & A4039 , 3: ST_CON
         IF $TIMER_FLAG[8] AND NOT $FLAG[325] AND NOT $FLAG[329] AND $OUT[4039] THEN
            PREVSTEP = $APP_INT[5]
            $APP_INT[5] = 67
         ENDIF
      ;ENDFOLD
   ;ENDFOLD
   ;FOLD SCHRITT 67 -- STAT EZ1/SP1/KE1 -- ;%{P}%MKUKATPVW,%CSTEP,%VST_NR,%P 1:SCHRITT, 2:67, 3: STAT EZ1/SP1/KE1
      ;FOLD ;%{H}
         Case 67
      ;ENDFOLD
      ;FOLD -- Hilfsflag SK Programmwechsel -- ;%{SE}%MKUKATPVW %CVW_COM %VCOMMENT %P 2:-- Hilfsflag SK Programmwechsel --, 3: VW_COMMENT
      ;ENDFOLD
      ;FOLD F334 = AUS ;%{SE}%MKUKATPVW %CVW_SPS %VBOASG %P 2:F334 = AUS, 3: BOASG
         $FLAG[334] = FALSE
      ;ENDFOLD
      ;FOLD -- Quitt. Fraesen SK1 -- ;%{SE}%MKUKATPVW %CVW_COM %VCOMMENT %P 2:-- Quitt. Fraesen SK1 --, 3: VW_COMMENT
      ;ENDFOLD
      ;FOLD A786 = (!F329 & !F322 & !F830) + (F830 & A786) ;%{SE}%MKUKATPVW %CVW_SPS %VBOASG %P 2:A786 = (!F329 & !F322 & !F830) + (F830 & A786), 3: BOASG
         $OUT[786] = (NOT $FLAG[329] AND NOT $FLAG[322] AND NOT $FLAG[830]) OR ($FLAG[830] AND $OUT[786])
      ;ENDFOLD
      ;FOLD A722 = (!F329 & !F322 & F830) + (!F830 & A722) ;%{SE}%MKUKATPVW %CVW_SPS %VBOASG %P 2:A722 = (!F329 & !F322 & F830) + (!F830 & A722), 3: BOASG
         $OUT[722] = (NOT $FLAG[329] AND NOT $FLAG[322] AND $FLAG[830]) OR (NOT $FLAG[830] AND $OUT[722])
      ;ENDFOLD
      ;FOLD -- RSK Sammelstoerung -- ;%{SE}%MKUKATPVW %CVW_COM %VCOMMENT %P 2:-- RSK Sammelstoerung --, 3: VW_COMMENT
      ;ENDFOLD
      ;FOLD F329 = T9 ;%{SE}%MKUKATPVW %CVW_SPS %VBOASG %P 2:F329 = T9, 3: BOASG
         $FLAG[329] = $TIMER_FLAG[9]
      ;ENDFOLD
      ;FOLD -- Messen nach Fraesen -- ;%{SE}%MKUKATPVW %CVW_COM %VCOMMENT %P 2:-- Messen nach Fraesen --, 3: VW_COMMENT
      ;ENDFOLD
      ;FOLD A759 = (!F78 & F79 & !F830) + (F830 & A759) ;%{SE}%MKUKATPVW %CVW_SPS %VBOASG %P 2:A759 = (!F78 & F79 & !F830) + (F830 & A759), 3: BOASG
         $OUT[759] = (NOT $FLAG[78] AND $FLAG[79] AND NOT $FLAG[830]) OR ($FLAG[830] AND $OUT[759])
      ;ENDFOLD
      ;FOLD A758 = (F78 & !F79 & !F830) + (F830 & A758) ;%{SE}%MKUKATPVW %CVW_SPS %VBOASG %P 2:A758 = (F78 & !F79 & !F830) + (F830 & A758), 3: BOASG
         $OUT[758] = ($FLAG[78] AND NOT $FLAG[79] AND NOT $FLAG[830]) OR ($FLAG[830] AND $OUT[758])
      ;ENDFOLD
      ;FOLD F836 = (F78 + F79) & !F329 ;%{SE}%MKUKATPVW %CVW_SPS %VBOASG %P 2:F836 = (F78 + F79) & !F329, 3: BOASG
         $FLAG[836] = ($FLAG[78] OR $FLAG[79]) AND NOT $FLAG[329]
      ;ENDFOLD
      ;FOLD A757 = (F836 & !F830) + (F830 & A757) ;%{SE}%MKUKATPVW %CVW_SPS %VBOASG %P 2:A757 = (F836 & !F830) + (F830 & A757), 3: BOASG
         $OUT[757] = ($FLAG[836] AND NOT $FLAG[830]) OR ($FLAG[830] AND $OUT[757])
      ;ENDFOLD
      ;FOLD A725 = (F836 & F830) + (!F830 & A725) ;%{SE}%MKUKATPVW %CVW_SPS %VBOASG %P 2:A725 = (F836 & F830) + (!F830 & A725), 3: BOASG
         $OUT[725] = ($FLAG[836] AND $FLAG[830]) OR (NOT $FLAG[830] AND $OUT[725])
      ;ENDFOLD
      ;FOLD Schritt 68 = A4039 & (!E786 & E787 & !E788 & !F830) + (!E722 & E724 & !E723 & F830)  ;%{SE}%MKUKATPVW %CVW_SPS %VST_CON %P 2:Schritt 68 = A4039 & (!E786 & E787 & !E788 & !F830) + (!E722 & E724 & !E723 & F830) , 3: ST_CON
         IF $OUT[4039] AND (NOT $IN[786] AND $IN[787] AND NOT $IN[788] AND NOT $FLAG[830]) OR (NOT $IN[722] AND $IN[724] AND NOT $IN[723] AND $FLAG[830]) THEN
            PREVSTEP = $APP_INT[5]
            $APP_INT[5] = 68
         ENDIF
      ;ENDFOLD
   ;ENDFOLD
   ;FOLD SCHRITT 68 -- STAT EZ1/SP1/KE1 -- ;%{P}%MKUKATPVW,%CSTEP,%VST_NR,%P 1:SCHRITT, 2:68, 3: STAT EZ1/SP1/KE1
      ;FOLD ;%{H}
         Case 68
      ;ENDFOLD
      ;FOLD F836 = AUS ;%{SE}%MKUKATPVW %CVW_SPS %VBOASG %P 2:F836 = AUS, 3: BOASG
         $FLAG[836] = FALSE
      ;ENDFOLD
      ;FOLD -- Hilfsflag SK Programmwechsel -- ;%{SE}%MKUKATPVW %CVW_COM %VCOMMENT %P 2:-- Hilfsflag SK Programmwechsel --, 3: VW_COMMENT
      ;ENDFOLD
      ;FOLD F334 = AUS ;%{SE}%MKUKATPVW %CVW_SPS %VBOASG %P 2:F334 = AUS, 3: BOASG
         $FLAG[334] = FALSE
      ;ENDFOLD
      ;FOLD -- RSK Sammelstoerung -- ;%{SE}%MKUKATPVW %CVW_COM %VCOMMENT %P 2:-- RSK Sammelstoerung --, 3: VW_COMMENT
      ;ENDFOLD
      ;FOLD F329 = T9 ;%{SE}%MKUKATPVW %CVW_SPS %VBOASG %P 2:F329 = T9, 3: BOASG
         $FLAG[329] = $TIMER_FLAG[9]
      ;ENDFOLD
      ;FOLD Schritt 69 =  A4039 & E717 & (E757 & !E776 & !F830 + T9) + (E725 & E726 & F830 + T9)  ;%{SE}%MKUKATPVW %CVW_SPS %VST_CON %P 2:Schritt 69 =  A4039 & E717 & (E757 & !E776 & !F830 + T9) + (E725 & E726 & F830 + T9) , 3: ST_CON
         IF $OUT[4039] AND $IN[717] AND ($IN[757] AND NOT $IN[776] AND NOT $FLAG[830] OR $TIMER_FLAG[9]) OR ($IN[725] AND $IN[726] AND $FLAG[830] OR $TIMER_FLAG[9]) THEN
            PREVSTEP = $APP_INT[5]
            $APP_INT[5] = 69
         ENDIF
      ;ENDFOLD
   ;ENDFOLD
   ;FOLD SCHRITT 69 -- STAT EZ1/SP1/KE1-- ;%{P}%MKUKATPVW,%CSTEP,%VST_NR,%P 1:SCHRITT, 2:69, 3: STAT EZ1/SP1/KE1
      ;FOLD ;%{H}
         Case 69
      ;ENDFOLD
      ;FOLD -- RSK Fehlerausgabe Kappenverschleiss -- ;%{SE}%MKUKATPVW %CVW_COM %VCOMMENT %P 2:-- RSK Fehlerausgabe Kappenverschleiss --, 3: VW_COMMENT
      ;ENDFOLD
      ;FOLD F122 = E777 ;%{SE}%MKUKATPVW %CVW_SPS %VBOASG %P 2:F122 = E777, 3: BOASG
         $FLAG[122] = $IN[777]
      ;ENDFOLD
      ;FOLD -- RSK Fehlerausgabe Messen -- ;%{SE}%MKUKATPVW %CVW_COM %VCOMMENT %P 2:-- RSK Fehlerausgabe Messen --, 3: VW_COMMENT
      ;ENDFOLD
      ;FOLD F326 = E776 + E777 + E778 + F326 ;%{SE}%MKUKATPVW %CVW_SPS %VBOASG %P 2:F326 = E776 + E777 + E778 + F326, 3: BOASG
         $FLAG[326] = $IN[776] OR $IN[777] OR $IN[778] OR $FLAG[326]
      ;ENDFOLD
      ;FOLD -- RSK Sammelstoerung -- ;%{SE}%MKUKATPVW %CVW_COM %VCOMMENT %P 2:-- RSK Sammelstoerung --, 3: VW_COMMENT
      ;ENDFOLD
      ;FOLD F329 = F326 ;%{SE}%MKUKATPVW %CVW_SPS %VBOASG %P 2:F329 = F326, 3: BOASG
         $FLAG[329] = $FLAG[326]
      ;ENDFOLD
      ;FOLD A758 = F830 & A758 ;%{SE}%MKUKATPVW %CVW_SPS %VBOASG %P 2:A758 = F830 & A758, 3: BOASG
         $OUT[758] = $FLAG[830] AND $OUT[758]
      ;ENDFOLD
      ;FOLD A759 = F830 & A759 ;%{SE}%MKUKATPVW %CVW_SPS %VBOASG %P 2:A759 = F830 & A759, 3: BOASG
         $OUT[759] = $FLAG[830] AND $OUT[759]
      ;ENDFOLD
      ;FOLD -- Ueberwachungszeit EZ1/SP1/KE1 Setzhub 2 -- ;%{SE}%MKUKATPVW %CVW_COM %VCOMMENT %P 2:-- Ueberwachungszeit EZ1/SP1/KE1 Setzhub 2 --, 3: VW_COMMENT
      ;ENDFOLD
      ;FOLD t9 ( EIN ) = -80[1/10Sek] ;%{SE}%MKUKATPVW %CVW_SPS %VTASG %P 2:t9 ( EIN ) = -80[1/10Sek], 3: TASG
         VW(#SET_TIME,TRUE,9,0,-80)
      ;ENDFOLD
      ;FOLD -- Druckvorgabe SK1/EZ1/SP1/KE1 -- ;%{SE}%MKUKATPVW %CVW_COM %VCOMMENT %P 2:-- Druckvorgabe SK1/EZ1/SP1/KE1 --, 3: VW_COMMENT
      ;ENDFOLD
      ;FOLD bin1 ( F78 ) = 41 ;%{SE}%MKUKATPVW %CVW_SPS %VARIASG %P 2:bin1 ( F78 ) = 41, 3: ARIASG
         VW(#BINOUT,$FLAG[78],1,41)
      ;ENDFOLD
      ;FOLD bin1 ( F79 ) = 51 ;%{SE}%MKUKATPVW %CVW_SPS %VARIASG %P 2:bin1 ( F79 ) = 51, 3: ARIASG
         VW(#BINOUT,$FLAG[79],1,51)
      ;ENDFOLD
      ;FOLD bin3 ( F78 ) = 41 ;%{SE}%MKUKATPVW %CVW_SPS %VARIASG %P 2:bin3 ( F78 ) = 41, 3: ARIASG
         VW(#BINOUT,$FLAG[78],3,41)
      ;ENDFOLD
      ;FOLD bin3 ( F79 ) = 51 ;%{SE}%MKUKATPVW %CVW_SPS %VARIASG %P 2:bin3 ( F79 ) = 51, 3: ARIASG
         VW(#BINOUT,$FLAG[79],3,51)
      ;ENDFOLD
      ;FOLD -- Wartezeit Programmwechsel SK -- ;%{SE}%MKUKATPVW %CVW_COM %VCOMMENT %P 2:-- Wartezeit Programmwechsel SK --, 3: VW_COMMENT
      ;ENDFOLD
      ;FOLD T8 ( !F334 ) = -2[1/10Sek] ;%{SE}%MKUKATPVW %CVW_SPS %VTASG %P 2:T8 ( !F334 ) = -2[1/10Sek], 3: TASG
         VW(#SET_TIME,NOT $FLAG[334],8,0,-2)
      ;ENDFOLD
      ;FOLD -- Hilfsflag SK Programmwechsel -- ;%{SE}%MKUKATPVW %CVW_COM %VCOMMENT %P 2:-- Hilfsflag SK Programmwechsel --, 3: VW_COMMENT
      ;ENDFOLD
      ;FOLD F334 = EIN ;%{SE}%MKUKATPVW %CVW_SPS %VBOASG %P 2:F334 = EIN, 3: BOASG
         $FLAG[334] = TRUE
      ;ENDFOLD
      ;FOLD Schritt 70 = T8 & !F335 & A4039  ;%{SE}%MKUKATPVW %CVW_SPS %VST_CON %P 2:Schritt 70 = T8 & !F335 & A4039 , 3: ST_CON
         IF $TIMER_FLAG[8] AND NOT $FLAG[335] AND $OUT[4039] THEN
            PREVSTEP = $APP_INT[5]
            $APP_INT[5] = 70
         ENDIF
      ;ENDFOLD
      ;FOLD Schritt 70 = T8 & F335 & !F78 & A4039  ;%{SE}%MKUKATPVW %CVW_SPS %VST_CON %P 2:Schritt 70 = T8 & F335 & !F78 & A4039 , 3: ST_CON
         IF $TIMER_FLAG[8] AND $FLAG[335] AND NOT $FLAG[78] AND $OUT[4039] THEN
            PREVSTEP = $APP_INT[5]
            $APP_INT[5] = 70
         ENDIF
      ;ENDFOLD
      ;FOLD Schritt 217 = T8 & F335 & F78 & A4039  ;%{SE}%MKUKATPVW %CVW_SPS %VST_CON %P 2:Schritt 217 = T8 & F335 & F78 & A4039 , 3: ST_CON
         IF $TIMER_FLAG[8] AND $FLAG[335] AND $FLAG[78] AND $OUT[4039] THEN
            PREVSTEP = $APP_INT[5]
            $APP_INT[5] = 217
         ENDIF
      ;ENDFOLD
   ;ENDFOLD
   ;FOLD SCHRITT 70 -- STAT EZ1/SP1/KE1 -- ;%{P}%MKUKATPVW,%CSTEP,%VST_NR,%P 1:SCHRITT, 2:70, 3: STAT EZ1/SP1/KE1
      ;FOLD ;%{H}
         Case 70
      ;ENDFOLD
